LIN {X 0.009,Y -453.231,Z 340.561,A 0.000,B 0.000,C 90.000,E1 100.894} C_DIS
LIN {X 0.062,Y -474.002,Z 340.550,A 0.000,B 0.000,C 90.000,E1 99.029} C_DIS
LIN {X 0.039,Y -492.580,Z 340.542,A 0.000,B 0.000,C 90.000,E1 97.530} C_DIS
LIN {X -0.190,Y -494.914,Z 340.541,A 0.000,B 0.000,C 90.000,E1 97.352} C_DIS
LIN {X 0.008,Y -496.686,Z 340.540,A 0.000,B 0.000,C 90.000,E1 97.125} C_DIS
LIN {X -0.081,Y -498.310,Z 340.538,A 0.000,B 0.000,C 90.000,E1 96.891} C_DIS
LIN {X -0.231,Y -499.526,Z 340.537,A 0.000,B 0.000,C 90.000,E1 96.663} C_DIS
LIN {X 0.045,Y -500.998,Z 340.534,A 0.000,B 0.000,C 90.000,E1 96.144} C_DIS
LIN {X -0.171,Y -501.409,Z 340.531,A 0.000,B 0.000,C 90.000,E1 95.682} C_DIS
LIN {X 0.120,Y -500.821,Z 340.529,A 0.000,B 0.000,C 90.000,E1 95.163} C_DIS
LIN {X -0.087,Y -499.136,Z 340.526,A 0.000,B 0.000,C 90.000,E1 94.702} C_DIS
LIN {X -0.213,Y -497.782,Z 340.525,A 0.000,B 0.000,C 90.000,E1 94.473} C_DIS
LIN {X -0.069,Y -492.467,Z 340.521,A 0.000,B 0.000,C 90.000,E1 93.726} C_DIS
LIN {X -0.123,Y -484.683,Z 340.515,A 0.000,B 0.000,C 90.000,E1 92.751} C_DIS
LIN {X 0.233,Y -466.512,Z 340.503,A 0.000,B 0.000,C 90.000,E1 90.458} C_DIS
LIN {X 0.098,Y -445.860,Z 340.487,A 0.000,B 0.000,C 90.000,E1 87.650} C_DIS
LIN {X -0.176,Y -427.360,Z 340.471,A 0.000,B 0.000,C 90.000,E1 84.780} C_DIS
LIN {X 0.063,Y -409.042,Z 340.453,A 0.000,B 0.000,C 90.000,E1 81.489} C_DIS
LIN {X 0.021,Y -396.047,Z 340.439,A 0.000,B 0.000,C 90.000,E1 78.993} C_DIS
LIN {X 0.024,Y -387.321,Z 340.429,A 0.000,B 0.000,C 90.000,E1 77.297} C_DIS
LIN {X 0.089,Y -374.251,Z 340.415,A 0.000,B 0.000,C 90.000,E1 74.700} C_DIS
LIN {X -0.037,Y -364.049,Z 340.404,A 0.000,B 0.000,C 90.000,E1 72.670} C_DIS
LIN {X -0.149,Y -353.844,Z 340.392,A 0.000,B 0.000,C 90.000,E1 70.604} C_DIS
LIN {X 0.016,Y -340.830,Z 340.377,A 0.000,B 0.000,C 90.000,E1 67.847} C_DIS
LIN {X 0.116,Y -331.356,Z 340.365,A 0.000,B 0.000,C 90.000,E1 65.665} C_DIS
LIN {X -0.087,Y -318.001,Z 340.346,A 0.000,B 0.000,C 90.000,E1 62.231} C_DIS
LIN {X -0.032,Y -306.589,Z 340.328,A 0.000,B 0.000,C 90.000,E1 58.997} C_DIS
LIN {X -0.090,Y -295.955,Z 340.309,A 0.000,B 0.000,C 90.000,E1 55.722} C_DIS
LIN {X 0.040,Y -286.100,Z 340.291,A 0.000,B 0.000,C 90.000,E1 52.351} C_DIS
LIN {X 0.082,Y -278.584,Z 340.276,A 0.000,B 0.000,C 90.000,E1 49.622} C_DIS
LIN {X 0.101,Y -272.888,Z 340.264,A 0.000,B 0.000,C 90.000,E1 47.553} C_DIS
LIN {X 0.135,Y -265.279,Z 340.249,A 0.000,B 0.000,C 90.000,E1 44.757} C_DIS
LIN {X -0.099,Y -259.648,Z 340.237,A 0.000,B 0.000,C 90.000,E1 42.690} C_DIS
LIN {X -0.055,Y -253.941,Z 340.225,A 0.000,B 0.000,C 90.000,E1 40.539} C_DIS
LIN {X -0.091,Y -248.138,Z 340.213,A 0.000,B 0.000,C 90.000,E1 38.382} C_DIS
LIN {X -0.010,Y -240.251,Z 340.197,A 0.000,B 0.000,C 90.000,E1 35.438} C_DIS
LIN {X -0.017,Y -232.499,Z 340.180,A 0.000,B 0.000,C 90.000,E1 32.467} C_DIS
LIN {X -0.049,Y -223.369,Z 340.159,A 0.000,B 0.000,C 90.000,E1 28.693} C_DIS
LIN {X 0.043,Y -216.611,Z 340.142,A 0.000,B 0.000,C 90.000,E1 25.591} C_DIS
LIN {X 0.076,Y -210.503,Z 340.125,A 0.000,B 0.000,C 90.000,E1 22.461} C_DIS
LIN {X -0.008,Y -205.261,Z 340.107,A 0.000,B 0.000,C 90.000,E1 19.322} C_DIS
LIN {X 0.011,Y -199.604,Z 340.085,A 0.000,B 0.000,C 90.000,E1 15.315} C_DIS
LIN {X 0.091,Y -195.082,Z 340.063,A 0.000,B 0.000,C 90.000,E1 11.243} C_DIS
LIN {X -0.003,Y -191.668,Z 340.040,A 0.000,B 0.000,C 90.000,E1 7.182} C_DIS
LIN {X -0.072,Y -188.853,Z 340.008,A 0.000,B 0.000,C 90.000,E1 1.432} C_DIS
LIN {X 0.006,Y -189.839,Z 339.938,A 0.000,B 0.000,C 90.000,E1 348.757} C_DIS
LIN {X 0.053,Y -192.868,Z 339.910,A 0.000,B 0.000,C 90.000,E1 343.795} C_DIS
LIN {X 0.056,Y -196.554,Z 339.887,A 0.000,B 0.000,C 90.000,E1 339.699} C_DIS
LIN {X -0.036,Y -201.292,Z 339.865,A 0.000,B 0.000,C 90.000,E1 335.665} C_DIS
LIN {X -0.008,Y -207.084,Z 339.842,A 0.000,B 0.000,C 90.000,E1 331.641} C_DIS
LIN {X 0.024,Y -212.411,Z 339.825,A 0.000,B 0.000,C 90.000,E1 328.456} C_DIS
LIN {X -0.067,Y -219.844,Z 339.803,A 0.000,B 0.000,C 90.000,E1 324.562} C_DIS
LIN {X 0.043,Y -227.918,Z 339.782,A 0.000,B 0.000,C 90.000,E1 320.678} C_DIS
LIN {X -0.140,Y -236.318,Z 339.763,A 0.000,B 0.000,C 90.000,E1 317.310} C_DIS
LIN {X -0.079,Y -245.981,Z 339.744,A 0.000,B 0.000,C 90.000,E1 313.947} C_DIS
LIN {X 0.128,Y -256.915,Z 339.726,A 0.000,B 0.000,C 90.000,E1 310.620} C_DIS
LIN {X -0.016,Y -268.632,Z 339.708,A 0.000,B 0.000,C 90.000,E1 307.443} C_DIS
LIN {X -0.052,Y -280.119,Z 339.693,A 0.000,B 0.000,C 90.000,E1 304.659} C_DIS
LIN {X -0.018,Y -291.107,Z 339.679,A 0.000,B 0.000,C 90.000,E1 302.260} C_DIS
LIN {X -0.158,Y -306.784,Z 339.663,A 0.000,B 0.000,C 90.000,E1 299.283} C_DIS
LIN {X -0.051,Y -318.097,Z 339.652,A 0.000,B 0.000,C 90.000,E1 297.308} C_DIS
LIN {X -0.013,Y -339.341,Z 339.634,A 0.000,B 0.000,C 90.000,E1 294.131} C_DIS
LIN {X 0.012,Y -352.717,Z 339.624,A 0.000,B 0.000,C 90.000,E1 292.280} C_DIS
LIN {X -0.103,Y -375.772,Z 339.607,A 0.000,B 0.000,C 90.000,E1 289.322} C_DIS
LIN {X 0.153,Y -395.779,Z 339.594,A 0.000,B 0.000,C 90.000,E1 286.985} C_DIS
LIN {X 0.143,Y -408.300,Z 339.587,A 0.000,B 0.000,C 90.000,E1 285.607} C_DIS
LIN {X -0.126,Y -423.347,Z 339.578,A 0.000,B 0.000,C 90.000,E1 284.008} C_DIS
LIN {X 0.082,Y -430.579,Z 339.573,A 0.000,B 0.000,C 90.000,E1 283.175} C_DIS
LIN {X 0.206,Y -437.414,Z 339.569,A 0.000,B 0.000,C 90.000,E1 282.355} C_DIS
LIN {X 0.175,Y -445.719,Z 339.563,A 0.000,B 0.000,C 90.000,E1 281.299} C_DIS
LIN {X 0.156,Y -453.343,Z 339.557,A 0.000,B 0.000,C 90.000,E1 280.254} C_DIS
LIN {X -0.223,Y -460.409,Z 339.551,A 0.000,B 0.000,C 90.000,E1 279.265} C_DIS
LIN {X 0.159,Y -468.590,Z 339.544,A 0.000,B 0.000,C 90.000,E1 277.936} C_DIS
LIN {X -0.059,Y -474.516,Z 339.539,A 0.000,B 0.000,C 90.000,E1 276.947} C_DIS
LIN {X 0.199,Y -479.773,Z 339.533,A 0.000,B 0.000,C 90.000,E1 275.910} C_DIS
LIN {X -0.127,Y -482.067,Z 339.530,A 0.000,B 0.000,C 90.000,E1 275.448} C_DIS
LIN {X -0.003,Y -484.044,Z 339.527,A 0.000,B 0.000,C 90.000,E1 274.935} C_DIS
LIN {X 0.172,Y -485.593,Z 339.525,A 0.000,B 0.000,C 90.000,E1 274.416} C_DIS
LIN {X -0.129,Y -486.743,Z 339.522,A 0.000,B 0.000,C 90.000,E1 273.955} C_DIS
LIN {X 0.031,Y -487.515,Z 339.519,A 0.000,B 0.000,C 90.000,E1 273.440} C_DIS
LIN {X 0.229,Y -487.879,Z 339.516,A 0.000,B 0.000,C 90.000,E1 272.922} C_DIS
LIN {X -0.083,Y -487.951,Z 339.514,A 0.000,B 0.000,C 90.000,E1 272.465} C_DIS
LIN {X -0.193,Y -487.478,Z 339.508,A 0.000,B 0.000,C 90.000,E1 271.489} C_DIS
LIN {X -0.012,Y -486.912,Z 339.505,A 0.000,B 0.000,C 90.000,E1 270.974} C_DIS
LIN {X 0.167,Y -486.115,Z 339.503,A 0.000,B 0.000,C 90.000,E1 270.458} C_DIS
LIN {X -0.142,Y -484.938,Z 339.500,A 0.000,B 0.000,C 90.000,E1 270.000} C_DIS
LIN {X 0.030,Y -483.269,Z 339.497,A 0.000,B 0.000,C 90.000,E1 269.484} C_DIS
LIN {X -0.129,Y -482.227,Z 339.496,A 0.000,B 0.000,C 90.000,E1 269.255} C_DIS
LIN {X 0.026,Y -479.578,Z 339.493,A 0.000,B 0.000,C 90.000,E1 268.740} C_DIS
LIN {X 0.163,Y -476.054,Z 339.490,A 0.000,B 0.000,C 90.000,E1 268.224} C_DIS
LIN {X 0.006,Y -473.958,Z 339.489,A 0.000,B 0.000,C 90.000,E1 267.993} C_DIS
LIN {X 0.114,Y -468.786,Z 339.486,A 0.000,B 0.000,C 90.000,E1 267.478} C_DIS
LIN {X 0.067,Y -465.947,Z 339.485,A 0.000,B 0.000,C 90.000,E1 267.249} C_DIS
LIN {X -0.155,Y -459.544,Z 339.482,A 0.000,B 0.000,C 90.000,E1 266.846} C_DIS
LIN {X 0.221,Y -452.496,Z 339.480,A 0.000,B 0.000,C 90.000,E1 266.445} C_DIS
LIN {X -0.155,Y -445.052,Z 339.479,A 0.000,B 0.000,C 90.000,E1 266.216} C_DIS
LIN {X -0.036,Y -437.239,Z 339.478,A 0.000,B 0.000,C 90.000,E1 265.988} C_DIS
LIN {X 0.127,Y -428.216,Z 339.477,A 0.000,B 0.000,C 90.000,E1 265.812} C_DIS
LIN {X 0.103,Y -421.480,Z 339.477,A 0.000,B 0.000,C 90.000,E1 265.755} C_DIS
LIN {X -0.019,Y -417.651,Z 339.476,A 0.000,B 0.000,C 90.000,E1 265.755} C_DIS
LIN {X -0.034,Y -180.912,Z 339.476,A 0.000,B 0.000,C 90.000,E1 265.755} C_DIS
LIN {X 0.074,Y -180.824,Z 339.471,A 0.000,B 0.000,C 90.000,E1 264.837} C_DIS
LIN {X -0.026,Y -178.929,Z 339.443,A 0.000,B 0.000,C 90.000,E1 259.803} C_DIS
LIN {X 0.012,Y -175.976,Z 339.415,A 0.000,B 0.000,C 90.000,E1 254.700} C_DIS
LIN {X -0.043,Y -175.465,Z 339.410,A 0.000,B 0.000,C 90.000,E1 253.866} C_DIS
LIN {X 0.014,Y -172.215,Z 339.387,A 0.000,B 0.000,C 90.000,E1 249.571} C_DIS
LIN {X -0.009,Y -171.691,Z 339.382,A 0.000,B 0.000,C 90.000,E1 248.720} C_DIS
LIN {X -0.019,Y -167.917,Z 339.358,A 0.000,B 0.000,C 90.000,E1 244.409} C_DIS
LIN {X -0.001,Y -166.660,Z 339.348,A 0.000,B 0.000,C 90.000,E1 242.666} C_DIS
LIN {X -0.084,Y -162.643,Z 339.324,A 0.000,B 0.000,C 90.000,E1 238.329} C_DIS
LIN {X -0.022,Y -161.331,Z 339.314,A 0.000,B 0.000,C 90.000,E1 236.548} C_DIS
LIN {X 0.021,Y -157.327,Z 339.290,A 0.000,B 0.000,C 90.000,E1 232.110} C_DIS
LIN {X -0.045,Y -155.308,Z 339.275,A 0.000,B 0.000,C 90.000,E1 229.461} C_DIS
LIN {X -0.007,Y -151.666,Z 339.250,A 0.000,B 0.000,C 90.000,E1 224.960} C_DIS
LIN {X 0.037,Y -150.532,Z 339.240,A 0.000,B 0.000,C 90.000,E1 223.137} C_DIS
LIN {X -0.033,Y -147.257,Z 339.215,A 0.000,B 0.000,C 90.000,E1 218.624} C_DIS
LIN {X 0.024,Y -145.283,Z 339.194,A 0.000,B 0.000,C 90.000,E1 214.945} C_DIS
LIN {X 0.058,Y -142.385,Z 339.164,A 0.000,B 0.000,C 90.000,E1 209.411} C_DIS
LIN {X -0.020,Y -141.362,Z 339.148,A 0.000,B 0.000,C 90.000,E1 206.668} C_DIS
LIN {X -0.042,Y -139.343,Z 339.112,A 0.000,B 0.000,C 90.000,E1 200.174} C_DIS
LIN {X -0.036,Y -139.012,Z 339.102,A 0.000,B 0.000,C 90.000,E1 198.308} C_DIS
LIN {X -0.041,Y -138.341,Z 339.055,A 0.000,B 0.000,C 90.000,E1 189.905} C_DIS
LIN {X -0.021,Y -139.398,Z 339.008,A 0.000,B 0.000,C 90.000,E1 181.489} C_DIS
LIN {X 0.032,Y -141.300,Z 338.972,A 0.000,B 0.000,C 90.000,E1 174.951} C_DIS
LIN {X -0.010,Y -142.662,Z 338.957,A 0.000,B 0.000,C 90.000,E1 172.186} C_DIS
LIN {X -0.061,Y -145.008,Z 338.931,A 0.000,B 0.000,C 90.000,E1 167.589} C_DIS
LIN {X -0.071,Y -147.634,Z 338.911,A 0.000,B 0.000,C 90.000,E1 163.921} C_DIS
LIN {X 0.007,Y -150.265,Z 338.890,A 0.000,B 0.000,C 90.000,E1 160.242} C_DIS
LIN {X 0.020,Y -153.664,Z 338.870,A 0.000,B 0.000,C 90.000,E1 156.613} C_DIS
LIN {X 0.076,Y -157.079,Z 338.850,A 0.000,B 0.000,C 90.000,E1 152.999} C_DIS
LIN {X 0.015,Y -161.214,Z 338.830,A 0.000,B 0.000,C 90.000,E1 149.459} C_DIS
LIN {X -0.037,Y -163.303,Z 338.821,A 0.000,B 0.000,C 90.000,E1 147.709} C_DIS
LIN {X -0.028,Y -167.752,Z 338.801,A 0.000,B 0.000,C 90.000,E1 144.196} C_DIS
LIN {X -0.009,Y -171.569,Z 338.787,A 0.000,B 0.000,C 90.000,E1 141.582} C_DIS
LIN {X -0.075,Y -176.516,Z 338.767,A 0.000,B 0.000,C 90.000,E1 138.162} C_DIS
LIN {X 0.050,Y -180.814,Z 338.753,A 0.000,B 0.000,C 90.000,E1 135.567} C_DIS
LIN {X 0.035,Y -186.222,Z 338.735,A 0.000,B 0.000,C 90.000,E1 132.204} C_DIS
LIN {X -0.027,Y -190.859,Z 338.721,A 0.000,B 0.000,C 90.000,E1 129.725} C_DIS
LIN {X 0.007,Y -196.621,Z 338.702,A 0.000,B 0.000,C 90.000,E1 126.423} C_DIS
LIN {X 0.100,Y -200.747,Z 338.691,A 0.000,B 0.000,C 90.000,E1 124.326} C_DIS
LIN {X 0.115,Y -300.828,Z 338.691,A 0.000,B 0.000,C 90.000,E1 124.326} C_DIS
LIN {X -0.175,Y -306.487,Z 338.690,A 0.000,B 0.000,C 90.000,E1 124.199} C_DIS
LIN {X -0.039,Y -308.951,Z 338.689,A 0.000,B 0.000,C 90.000,E1 123.992} C_DIS
LIN {X -0.176,Y -312.801,Z 338.686,A 0.000,B 0.000,C 90.000,E1 123.579} C_DIS
LIN {X -0.045,Y -314.697,Z 338.685,A 0.000,B 0.000,C 90.000,E1 123.245} C_DIS
LIN {X -0.176,Y -316.191,Z 338.683,A 0.000,B 0.000,C 90.000,E1 122.959} C_DIS
LIN {X 0.029,Y -329.310,Z 338.663,A 0.000,B 0.000,C 90.000,E1 119.411} C_DIS
LIN {X -0.078,Y -341.472,Z 338.648,A 0.000,B 0.000,C 90.000,E1 116.616} C_DIS
LIN {X -0.012,Y -353.536,Z 338.634,A 0.000,B 0.000,C 90.000,E1 114.155} C_DIS
LIN {X -0.113,Y -366.874,Z 338.621,A 0.000,B 0.000,C 90.000,E1 111.770} C_DIS
LIN {X 0.053,Y -381.582,Z 338.608,A 0.000,B 0.000,C 90.000,E1 109.396} C_DIS
LIN {X 0.113,Y -397.769,Z 338.595,A 0.000,B 0.000,C 90.000,E1 107.094} C_DIS
LIN {X -0.164,Y -415.556,Z 338.583,A 0.000,B 0.000,C 90.000,E1 104.898} C_DIS
LIN {X 0.040,Y -435.006,Z 338.571,A 0.000,B 0.000,C 90.000,E1 102.703} C_DIS
LIN {X -0.132,Y -455.300,Z 338.559,A 0.000,B 0.000,C 90.000,E1 100.715} C_DIS
LIN {X -0.032,Y -476.123,Z 338.549,A 0.000,B 0.000,C 90.000,E1 98.859} C_DIS
LIN {X 0.140,Y -494.540,Z 338.541,A 0.000,B 0.000,C 90.000,E1 97.352} C_DIS
LIN {X -0.157,Y -496.447,Z 338.540,A 0.000,B 0.000,C 90.000,E1 97.182} C_DIS
LIN {X 0.247,Y -498.182,Z 338.538,A 0.000,B 0.000,C 90.000,E1 96.891} C_DIS
LIN {X 0.097,Y -499.483,Z 338.537,A 0.000,B 0.000,C 90.000,E1 96.663} C_DIS
LIN {X -0.125,Y -501.090,Z 338.534,A 0.000,B 0.000,C 90.000,E1 96.201} C_DIS
LIN {X 0.159,Y -501.614,Z 338.532,A 0.000,B 0.000,C 90.000,E1 95.682} C_DIS
LIN {X -0.050,Y -501.141,Z 338.529,A 0.000,B 0.000,C 90.000,E1 95.220} C_DIS
LIN {X 0.241,Y -499.590,Z 338.526,A 0.000,B 0.000,C 90.000,E1 94.702} C_DIS
LIN {X 0.116,Y -498.324,Z 338.525,A 0.000,B 0.000,C 90.000,E1 94.473} C_DIS
LIN {X -0.231,Y -493.062,Z 338.521,A 0.000,B 0.000,C 90.000,E1 93.784} C_DIS
LIN {X 0.207,Y -485.329,Z 338.515,A 0.000,B 0.000,C 90.000,E1 92.751} C_DIS
LIN {X 0.101,Y -467.113,Z 338.503,A 0.000,B 0.000,C 90.000,E1 90.516} C_DIS
LIN {X -0.010,Y -446.408,Z 338.487,A 0.000,B 0.000,C 90.000,E1 87.707} C_DIS
LIN {X 0.164,Y -427.828,Z 338.471,A 0.000,B 0.000,C 90.000,E1 84.780} C_DIS
LIN {X 0.000,Y -409.501,Z 338.453,A 0.000,B 0.000,C 90.000,E1 81.546} C_DIS
LIN {X -0.025,Y -396.518,Z 338.439,A 0.000,B 0.000,C 90.000,E1 79.050} C_DIS
LIN {X -0.011,Y -387.800,Z 338.430,A 0.000,B 0.000,C 90.000,E1 77.353} C_DIS
LIN {X 0.072,Y -374.714,Z 338.415,A 0.000,B 0.000,C 90.000,E1 74.755} C_DIS
LIN {X -0.040,Y -364.517,Z 338.404,A 0.000,B 0.000,C 90.000,E1 72.725} C_DIS
LIN {X 0.195,Y -354.305,Z 338.392,A 0.000,B 0.000,C 90.000,E1 70.604} C_DIS
LIN {X -0.083,Y -341.288,Z 338.377,A 0.000,B 0.000,C 90.000,E1 67.922} C_DIS
LIN {X 0.022,Y -331.789,Z 338.365,A 0.000,B 0.000,C 90.000,E1 65.741} C_DIS
LIN {X -0.023,Y -318.435,Z 338.346,A 0.000,B 0.000,C 90.000,E1 62.281} C_DIS
LIN {X -0.064,Y -305.897,Z 338.326,A 0.000,B 0.000,C 90.000,E1 58.742} C_DIS
LIN {X 0.031,Y -294.336,Z 338.306,A 0.000,B 0.000,C 90.000,E1 55.102} C_DIS
LIN {X 0.049,Y -284.581,Z 338.288,A 0.000,B 0.000,C 90.000,E1 51.743} C_DIS
LIN {X 0.057,Y -277.079,Z 338.272,A 0.000,B 0.000,C 90.000,E1 49.013} C_DIS
LIN {X 0.048,Y -271.336,Z 338.261,A 0.000,B 0.000,C 90.000,E1 46.944} C_DIS
LIN {X -0.146,Y -263.784,Z 338.245,A 0.000,B 0.000,C 90.000,E1 44.190} C_DIS
LIN {X 0.047,Y -256.224,Z 338.230,A 0.000,B 0.000,C 90.000,E1 41.310} C_DIS
LIN {X -0.138,Y -250.470,Z 338.218,A 0.000,B 0.000,C 90.000,E1 39.197} C_DIS
LIN {X -0.047,Y -244.568,Z 338.205,A 0.000,B 0.000,C 90.000,E1 36.996} C_DIS
LIN {X -0.007,Y -236.727,Z 338.189,A 0.000,B 0.000,C 90.000,E1 34.040} C_DIS
LIN {X 0.124,Y -227.275,Z 338.168,A 0.000,B 0.000,C 90.000,E1 30.256} C_DIS
LIN {X -0.090,Y -218.546,Z 338.147,A 0.000,B 0.000,C 90.000,E1 26.488} C_DIS
LIN {X 0.082,Y -212.229,Z 338.130,A 0.000,B 0.000,C 90.000,E1 23.334} C_DIS
LIN {X 0.045,Y -206.750,Z 338.112,A 0.000,B 0.000,C 90.000,E1 20.194} C_DIS
LIN {X 0.043,Y -200.875,Z 338.090,A 0.000,B 0.000,C 90.000,E1 16.205} C_DIS
LIN {X -0.060,Y -196.971,Z 338.072,A 0.000,B 0.000,C 90.000,E1 13.008} C_DIS
LIN {X 0.006,Y -193.094,Z 338.050,A 0.000,B 0.000,C 90.000,E1 8.916} C_DIS
LIN {X -0.079,Y -189.956,Z 338.022,A 0.000,B 0.000,C 90.000,E1 4.012} C_DIS
LIN {X -0.027,Y -190.716,Z 337.928,A 0.000,B 0.000,C 90.000,E1 347.117} C_DIS
LIN {X -0.032,Y -194.238,Z 337.901,A 0.000,B 0.000,C 90.000,E1 342.181} C_DIS
LIN {X -0.046,Y -198.343,Z 337.878,A 0.000,B 0.000,C 90.000,E1 338.103} C_DIS
LIN {X 0.077,Y -203.519,Z 337.856,A 0.000,B 0.000,C 90.000,E1 334.024} C_DIS
LIN {X 0.003,Y -209.629,Z 337.834,A 0.000,B 0.000,C 90.000,E1 330.049} C_DIS
LIN {X 0.078,Y -216.752,Z 337.812,A 0.000,B 0.000,C 90.000,E1 326.087} C_DIS
LIN {X 0.143,Y -224.531,Z 337.790,A 0.000,B 0.000,C 90.000,E1 322.190} C_DIS
LIN {X -0.029,Y -231.488,Z 337.773,A 0.000,B 0.000,C 90.000,E1 319.175} C_DIS
LIN {X 0.085,Y -239.347,Z 337.756,A 0.000,B 0.000,C 90.000,E1 316.134} C_DIS
LIN {X -0.097,Y -249.498,Z 337.738,A 0.000,B 0.000,C 90.000,E1 312.852} C_DIS
LIN {X 0.041,Y -260.745,Z 337.720,A 0.000,B 0.000,C 90.000,E1 309.564} C_DIS
LIN {X 0.054,Y -272.865,Z 337.702,A 0.000,B 0.000,C 90.000,E1 306.377} C_DIS
LIN {X -0.072,Y -286.402,Z 337.685,A 0.000,B 0.000,C 90.000,E1 303.293} C_DIS
LIN {X -0.039,Y -301.568,Z 337.668,A 0.000,B 0.000,C 90.000,E1 300.256} C_DIS
LIN {X -0.080,Y -316.345,Z 337.653,A 0.000,B 0.000,C 90.000,E1 297.641} C_DIS
LIN {X -0.093,Y -337.413,Z 337.636,A 0.000,B 0.000,C 90.000,E1 294.463} C_DIS
LIN {X 0.034,Y -350.753,Z 337.626,A 0.000,B 0.000,C 90.000,E1 292.589} C_DIS
LIN {X 0.088,Y -368.997,Z 337.612,A 0.000,B 0.000,C 90.000,E1 290.174} C_DIS
LIN {X -0.144,Y -395.974,Z 337.595,A 0.000,B 0.000,C 90.000,E1 287.040} C_DIS
LIN {X 0.066,Y -408.645,Z 337.587,A 0.000,B 0.000,C 90.000,E1 285.607} C_DIS
LIN {X -0.243,Y -423.658,Z 337.578,A 0.000,B 0.000,C 90.000,E1 284.008} C_DIS
LIN {X -0.083,Y -430.903,Z 337.573,A 0.000,B 0.000,C 90.000,E1 283.175} C_DIS
LIN {X 0.040,Y -437.677,Z 337.569,A 0.000,B 0.000,C 90.000,E1 282.355} C_DIS
LIN {X 0.010,Y -445.911,Z 337.563,A 0.000,B 0.000,C 90.000,E1 281.299} C_DIS
LIN {X -0.011,Y -453.477,Z 337.557,A 0.000,B 0.000,C 90.000,E1 280.254} C_DIS
LIN {X 0.064,Y -460.491,Z 337.551,A 0.000,B 0.000,C 90.000,E1 279.208} C_DIS
LIN {X -0.010,Y -468.644,Z 337.544,A 0.000,B 0.000,C 90.000,E1 277.936} C_DIS
LIN {X 0.241,Y -474.530,Z 337.538,A 0.000,B 0.000,C 90.000,E1 276.891} C_DIS
LIN {X 0.027,Y -479.776,Z 337.533,A 0.000,B 0.000,C 90.000,E1 275.910} C_DIS
LIN {X 0.180,Y -482.032,Z 337.530,A 0.000,B 0.000,C 90.000,E1 275.391} C_DIS
LIN {X -0.177,Y -483.995,Z 337.527,A 0.000,B 0.000,C 90.000,E1 274.935} C_DIS
LIN {X -0.003,Y -485.531,Z 337.525,A 0.000,B 0.000,C 90.000,E1 274.416} C_DIS
LIN {X 0.181,Y -486.657,Z 337.522,A 0.000,B 0.000,C 90.000,E1 273.898} C_DIS
LIN {X -0.144,Y -487.374,Z 337.519,A 0.000,B 0.000,C 90.000,E1 273.440} C_DIS
LIN {X 0.052,Y -487.715,Z 337.516,A 0.000,B 0.000,C 90.000,E1 272.922} C_DIS
LIN {X 0.227,Y -487.811,Z 337.514,A 0.000,B 0.000,C 90.000,E1 272.407} C_DIS
LIN {X 0.115,Y -487.312,Z 337.508,A 0.000,B 0.000,C 90.000,E1 271.432} C_DIS
LIN {X -0.193,Y -486.761,Z 337.505,A 0.000,B 0.000,C 90.000,E1 270.974} C_DIS
LIN {X -0.014,Y -485.983,Z 337.503,A 0.000,B 0.000,C 90.000,E1 270.458} C_DIS
LIN {X 0.162,Y -484.816,Z 337.500,A 0.000,B 0.000,C 90.000,E1 269.943} C_DIS
LIN {X -0.151,Y -483.152,Z 337.497,A 0.000,B 0.000,C 90.000,E1 269.484} C_DIS
LIN {X 0.012,Y -480.854,Z 337.494,A 0.000,B 0.000,C 90.000,E1 268.969} C_DIS
LIN {X 0.157,Y -477.831,Z 337.492,A 0.000,B 0.000,C 90.000,E1 268.453} C_DIS
LIN {X -0.174,Y -473.839,Z 337.489,A 0.000,B 0.000,C 90.000,E1 267.993} C_DIS
LIN {X -0.065,Y -468.715,Z 337.486,A 0.000,B 0.000,C 90.000,E1 267.478} C_DIS
LIN {X -0.193,Y -462.406,Z 337.483,A 0.000,B 0.000,C 90.000,E1 267.020} C_DIS
LIN {X 0.077,Y -459.185,Z 337.482,A 0.000,B 0.000,C 90.000,E1 266.788} C_DIS
LIN {X -0.003,Y -452.049,Z 337.480,A 0.000,B 0.000,C 90.000,E1 266.445} C_DIS
LIN {X 0.085,Y -444.599,Z 337.479,A 0.000,B 0.000,C 90.000,E1 266.159} C_DIS
LIN {X -0.225,Y -436.603,Z 337.478,A 0.000,B 0.000,C 90.000,E1 265.988} C_DIS
LIN {X -0.027,Y -427.272,Z 337.477,A 0.000,B 0.000,C 90.000,E1 265.812} C_DIS
LIN {X -0.087,Y -417.710,Z 337.476,A 0.000,B 0.000,C 90.000,E1 265.755} C_DIS
LIN {X -0.062,Y -180.911,Z 337.476,A 0.000,B 0.000,C 90.000,E1 265.755} C_DIS
LIN {X 0.029,Y -180.820,Z 337.471,A 0.000,B 0.000,C 90.000,E1 264.837} C_DIS
LIN {X -0.071,Y -178.924,Z 337.443,A 0.000,B 0.000,C 90.000,E1 259.803} C_DIS
LIN {X -0.033,Y -175.970,Z 337.415,A 0.000,B 0.000,C 90.000,E1 254.700} C_DIS
LIN {X -0.038,Y -175.453,Z 337.410,A 0.000,B 0.000,C 90.000,E1 253.850} C_DIS
LIN {X -0.029,Y -172.206,Z 337.386,A 0.000,B 0.000,C 90.000,E1 249.571} C_DIS
LIN {X -0.052,Y -171.680,Z 337.382,A 0.000,B 0.000,C 90.000,E1 248.720} C_DIS
LIN {X -0.061,Y -167.906,Z 337.358,A 0.000,B 0.000,C 90.000,E1 244.409} C_DIS
LIN {X -0.042,Y -166.647,Z 337.348,A 0.000,B 0.000,C 90.000,E1 242.666} C_DIS
LIN {X 0.012,Y -162.631,Z 337.324,A 0.000,B 0.000,C 90.000,E1 238.280} C_DIS
LIN {X 0.071,Y -161.319,Z 337.314,A 0.000,B 0.000,C 90.000,E1 236.501} C_DIS
LIN {X -0.019,Y -157.315,Z 337.289,A 0.000,B 0.000,C 90.000,E1 232.110} C_DIS
LIN {X -0.086,Y -155.295,Z 337.275,A 0.000,B 0.000,C 90.000,E1 229.461} C_DIS
LIN {X 0.060,Y -151.655,Z 337.250,A 0.000,B 0.000,C 90.000,E1 224.919} C_DIS
LIN {X -0.003,Y -150.522,Z 337.240,A 0.000,B 0.000,C 90.000,E1 223.137} C_DIS
LIN {X 0.020,Y -147.247,Z 337.214,A 0.000,B 0.000,C 90.000,E1 218.588} C_DIS
LIN {X -0.015,Y -145.272,Z 337.194,A 0.000,B 0.000,C 90.000,E1 214.945} C_DIS
LIN {X 0.019,Y -142.379,Z 337.163,A 0.000,B 0.000,C 90.000,E1 209.411} C_DIS
LIN {X 0.069,Y -141.354,Z 337.148,A 0.000,B 0.000,C 90.000,E1 206.616} C_DIS
LIN {X 0.051,Y -139.340,Z 337.112,A 0.000,B 0.000,C 90.000,E1 200.120} C_DIS
LIN {X -0.030,Y -139.008,Z 337.102,A 0.000,B 0.000,C 90.000,E1 198.290} C_DIS
LIN {X 0.058,Y -138.340,Z 337.055,A 0.000,B 0.000,C 90.000,E1 189.849} C_DIS
LIN {X -0.059,Y -139.403,Z 337.008,A 0.000,B 0.000,C 90.000,E1 181.489} C_DIS
LIN {X -0.005,Y -141.308,Z 336.972,A 0.000,B 0.000,C 90.000,E1 174.951} C_DIS
LIN {X -0.048,Y -142.668,Z 336.956,A 0.000,B 0.000,C 90.000,E1 172.186} C_DIS
LIN {X 0.073,Y -145.017,Z 336.931,A 0.000,B 0.000,C 90.000,E1 167.521} C_DIS
LIN {X 0.031,Y -147.644,Z 336.910,A 0.000,B 0.000,C 90.000,E1 163.866} C_DIS
LIN {X -0.033,Y -150.277,Z 336.890,A 0.000,B 0.000,C 90.000,E1 160.242} C_DIS
LIN {X -0.021,Y -153.681,Z 336.870,A 0.000,B 0.000,C 90.000,E1 156.613} C_DIS
LIN {X 0.035,Y -157.095,Z 336.850,A 0.000,B 0.000,C 90.000,E1 152.999} C_DIS
LIN {X -0.026,Y -161.233,Z 336.830,A 0.000,B 0.000,C 90.000,E1 149.459} C_DIS
LIN {X 0.059,Y -163.321,Z 336.820,A 0.000,B 0.000,C 90.000,E1 147.661} C_DIS
LIN {X -0.070,Y -167.772,Z 336.801,A 0.000,B 0.000,C 90.000,E1 144.196} C_DIS
LIN {X 0.082,Y -171.588,Z 336.786,A 0.000,B 0.000,C 90.000,E1 141.537} C_DIS
LIN {X 0.012,Y -176.538,Z 336.767,A 0.000,B 0.000,C 90.000,E1 138.119} C_DIS
LIN {X 0.005,Y -180.837,Z 336.753,A 0.000,B 0.000,C 90.000,E1 135.567} C_DIS
LIN {X -0.010,Y -186.247,Z 336.734,A 0.000,B 0.000,C 90.000,E1 132.204} C_DIS
LIN {X -0.073,Y -190.883,Z 336.721,A 0.000,B 0.000,C 90.000,E1 129.725} C_DIS
LIN {X -0.040,Y -196.647,Z 336.702,A 0.000,B 0.000,C 90.000,E1 126.423} C_DIS
LIN {X 0.069,Y -200.850,Z 336.691,A 0.000,B 0.000,C 90.000,E1 124.278} C_DIS
LIN {X 0.071,Y -300.665,Z 336.691,A 0.000,B 0.000,C 90.000,E1 124.278} C_DIS
LIN {X 0.041,Y -301.580,Z 336.690,A 0.000,B 0.000,C 90.000,E1 124.278} C_DIS
LIN {X 0.051,Y -306.312,Z 336.690,A 0.000,B 0.000,C 90.000,E1 124.119} C_DIS
LIN {X -0.113,Y -308.604,Z 336.689,A 0.000,B 0.000,C 90.000,E1 123.992} C_DIS
LIN {X -0.110,Y -312.476,Z 336.686,A 0.000,B 0.000,C 90.000,E1 123.579} C_DIS
LIN {X 0.103,Y -314.402,Z 336.685,A 0.000,B 0.000,C 90.000,E1 123.245} C_DIS
LIN {X 0.053,Y -315.926,Z 336.683,A 0.000,B 0.000,C 90.000,E1 122.959} C_DIS
LIN {X -0.087,Y -318.377,Z 336.680,A 0.000,B 0.000,C 90.000,E1 122.339} C_DIS
LIN {X -0.025,Y -329.126,Z 336.664,A 0.000,B 0.000,C 90.000,E1 119.461} C_DIS
LIN {X 0.157,Y -341.266,Z 336.648,A 0.000,B 0.000,C 90.000,E1 116.616} C_DIS
LIN {X -0.095,Y -353.311,Z 336.634,A 0.000,B 0.000,C 90.000,E1 114.207} C_DIS
LIN {X 0.129,Y -366.627,Z 336.621,A 0.000,B 0.000,C 90.000,E1 111.770} C_DIS
LIN {X -0.061,Y -381.312,Z 336.608,A 0.000,B 0.000,C 90.000,E1 109.450} C_DIS
LIN {X -0.019,Y -397.475,Z 336.595,A 0.000,B 0.000,C 90.000,E1 107.149} C_DIS
LIN {X 0.088,Y -415.235,Z 336.583,A 0.000,B 0.000,C 90.000,E1 104.898} C_DIS
LIN {X -0.227,Y -434.661,Z 336.571,A 0.000,B 0.000,C 90.000,E1 102.771} C_DIS
LIN {X 0.108,Y -454.946,Z 336.560,A 0.000,B 0.000,C 90.000,E1 100.715} C_DIS
LIN {X 0.197,Y -475.762,Z 336.549,A 0.000,B 0.000,C 90.000,E1 98.859} C_DIS
LIN {X -0.129,Y -494.264,Z 336.541,A 0.000,B 0.000,C 90.000,E1 97.409} C_DIS
LIN {X 0.063,Y -496.288,Z 336.540,A 0.000,B 0.000,C 90.000,E1 97.182} C_DIS
LIN {X -0.018,Y -498.108,Z 336.539,A 0.000,B 0.000,C 90.000,E1 96.947} C_DIS
LIN {X -0.161,Y -499.473,Z 336.537,A 0.000,B 0.000,C 90.000,E1 96.720} C_DIS
LIN {X 0.113,Y -501.190,Z 336.535,A 0.000,B 0.000,C 90.000,E1 96.201} C_DIS
LIN {X -0.102,Y -501.805,Z 336.532,A 0.000,B 0.000,C 90.000,E1 95.739} C_DIS
LIN {X 0.189,Y -501.421,Z 336.529,A 0.000,B 0.000,C 90.000,E1 95.220} C_DIS
LIN {X -0.017,Y -499.977,Z 336.526,A 0.000,B 0.000,C 90.000,E1 94.759} C_DIS
LIN {X -0.141,Y -498.779,Z 336.525,A 0.000,B 0.000,C 90.000,E1 94.531} C_DIS
LIN {X 0.138,Y -495.405,Z 336.522,A 0.000,B 0.000,C 90.000,E1 94.012} C_DIS
LIN {X 0.227,Y -489.833,Z 336.518,A 0.000,B 0.000,C 90.000,E1 93.269} C_DIS
LIN {X 0.142,Y -481.806,Z 336.513,A 0.000,B 0.000,C 90.000,E1 92.293} C_DIS
LIN {X -0.204,Y -457.951,Z 336.496,A 0.000,B 0.000,C 90.000,E1 89.312} C_DIS
LIN {X 0.189,Y -443.344,Z 336.485,A 0.000,B 0.000,C 90.000,E1 87.192} C_DIS
LIN {X -0.015,Y -423.471,Z 336.467,A 0.000,B 0.000,C 90.000,E1 84.033} C_DIS
LIN {X -0.087,Y -408.443,Z 336.452,A 0.000,B 0.000,C 90.000,E1 81.319} C_DIS
LIN {X -0.076,Y -395.470,Z 336.438,A 0.000,B 0.000,C 90.000,E1 78.814} C_DIS
LIN {X -0.078,Y -386.754,Z 336.428,A 0.000,B 0.000,C 90.000,E1 77.117} C_DIS
LIN {X -0.025,Y -375.108,Z 336.416,A 0.000,B 0.000,C 90.000,E1 74.810} C_DIS
LIN {X -0.122,Y -364.921,Z 336.404,A 0.000,B 0.000,C 90.000,E1 72.779} C_DIS
LIN {X 0.011,Y -354.701,Z 336.393,A 0.000,B 0.000,C 90.000,E1 70.678} C_DIS
LIN {X -0.132,Y -341.692,Z 336.378,A 0.000,B 0.000,C 90.000,E1 67.975} C_DIS
LIN {X -0.012,Y -332.176,Z 336.366,A 0.000,B 0.000,C 90.000,E1 65.793} C_DIS
LIN {X -0.183,Y -318.805,Z 336.346,A 0.000,B 0.000,C 90.000,E1 62.359} C_DIS
LIN {X -0.099,Y -307.403,Z 336.328,A 0.000,B 0.000,C 90.000,E1 59.125} C_DIS
LIN {X 0.120,Y -296.744,Z 336.310,A 0.000,B 0.000,C 90.000,E1 55.801} C_DIS
LIN {X 0.035,Y -286.843,Z 336.292,A 0.000,B 0.000,C 90.000,E1 52.477} C_DIS
LIN {X 0.102,Y -279.279,Z 336.276,A 0.000,B 0.000,C 90.000,E1 49.747} C_DIS
LIN {X -0.044,Y -273.588,Z 336.265,A 0.000,B 0.000,C 90.000,E1 47.715} C_DIS
LIN {X 0.010,Y -265.960,Z 336.250,A 0.000,B 0.000,C 90.000,E1 44.919} C_DIS
LIN {X -0.033,Y -260.331,Z 336.238,A 0.000,B 0.000,C 90.000,E1 42.813} C_DIS
LIN {X 0.018,Y -254.639,Z 336.226,A 0.000,B 0.000,C 90.000,E1 40.663} C_DIS
LIN {X -0.011,Y -248.859,Z 336.214,A 0.000,B 0.000,C 90.000,E1 38.508} C_DIS
LIN {X 0.090,Y -242.920,Z 336.202,A 0.000,B 0.000,C 90.000,E1 36.297} C_DIS
LIN {X -0.045,Y -235.119,Z 336.185,A 0.000,B 0.000,C 90.000,E1 33.372} C_DIS
LIN {X 0.041,Y -225.781,Z 336.164,A 0.000,B 0.000,C 90.000,E1 29.589} C_DIS
LIN {X -0.010,Y -218.811,Z 336.147,A 0.000,B 0.000,C 90.000,E1 26.539} C_DIS
LIN {X -0.034,Y -212.473,Z 336.130,A 0.000,B 0.000,C 90.000,E1 23.439} C_DIS
LIN {X -0.071,Y -206.980,Z 336.113,A 0.000,B 0.000,C 90.000,E1 20.301} C_DIS
LIN {X -0.072,Y -201.085,Z 336.091,A 0.000,B 0.000,C 90.000,E1 16.315} C_DIS
LIN {X 0.019,Y -197.161,Z 336.073,A 0.000,B 0.000,C 90.000,E1 13.063} C_DIS
LIN {X 0.087,Y -193.284,Z 336.050,A 0.000,B 0.000,C 90.000,E1 8.973} C_DIS
LIN {X -0.008,Y -190.135,Z 336.023,A 0.000,B 0.000,C 90.000,E1 4.073} C_DIS
LIN {X 0.045,Y -188.423,Z 335.970,A 0.000,B 0.000,C 90.000,E1 354.546} C_DIS
LIN {X -0.019,Y -190.776,Z 335.928,A 0.000,B 0.000,C 90.000,E1 347.117} C_DIS
LIN {X -0.021,Y -194.277,Z 335.901,A 0.000,B 0.000,C 90.000,E1 342.181} C_DIS
LIN {X -0.035,Y -198.366,Z 335.878,A 0.000,B 0.000,C 90.000,E1 338.103} C_DIS
LIN {X 0.090,Y -203.535,Z 335.856,A 0.000,B 0.000,C 90.000,E1 334.024} C_DIS
LIN {X 0.018,Y -209.618,Z 335.834,A 0.000,B 0.000,C 90.000,E1 330.049} C_DIS
LIN {X 0.091,Y -216.720,Z 335.812,A 0.000,B 0.000,C 90.000,E1 326.087} C_DIS
LIN {X -0.022,Y -224.475,Z 335.790,A 0.000,B 0.000,C 90.000,E1 322.236} C_DIS
LIN {X -0.018,Y -231.427,Z 335.773,A 0.000,B 0.000,C 90.000,E1 319.175} C_DIS
LIN {X 0.096,Y -239.298,Z 335.756,A 0.000,B 0.000,C 90.000,E1 316.134} C_DIS
LIN {X -0.086,Y -249.501,Z 335.738,A 0.000,B 0.000,C 90.000,E1 312.852} C_DIS
LIN {X 0.054,Y -260.771,Z 335.720,A 0.000,B 0.000,C 90.000,E1 309.564} C_DIS
LIN {X 0.068,Y -272.946,Z 335.702,A 0.000,B 0.000,C 90.000,E1 306.377} C_DIS
LIN {X -0.013,Y -284.958,Z 335.687,A 0.000,B 0.000,C 90.000,E1 303.627} C_DIS
LIN {X -0.016,Y -294.798,Z 335.676,A 0.000,B 0.000,C 90.000,E1 301.592} C_DIS
LIN {X -0.047,Y -310.859,Z 335.659,A 0.000,B 0.000,C 90.000,E1 298.615} C_DIS
LIN {X -0.075,Y -320.605,Z 335.650,A 0.000,B 0.000,C 90.000,E1 297.001} C_DIS
LIN {X 0.062,Y -339.905,Z 335.634,A 0.000,B 0.000,C 90.000,E1 294.131} C_DIS
LIN {X 0.100,Y -353.264,Z 335.624,A 0.000,B 0.000,C 90.000,E1 292.280} C_DIS
LIN {X -0.164,Y -374.040,Z 335.609,A 0.000,B 0.000,C 90.000,E1 289.631} C_DIS
LIN {X -0.097,Y -396.212,Z 335.595,A 0.000,B 0.000,C 90.000,E1 287.040} C_DIS
LIN {X 0.133,Y -408.808,Z 335.587,A 0.000,B 0.000,C 90.000,E1 285.607} C_DIS
LIN {X -0.177,Y -423.733,Z 335.578,A 0.000,B 0.000,C 90.000,E1 284.008} C_DIS
LIN {X -0.023,Y -430.972,Z 335.573,A 0.000,B 0.000,C 90.000,E1 283.175} C_DIS
LIN {X 0.101,Y -437.701,Z 335.569,A 0.000,B 0.000,C 90.000,E1 282.355} C_DIS
LIN {X 0.073,Y -445.896,Z 335.563,A 0.000,B 0.000,C 90.000,E1 281.299} C_DIS
LIN {X 0.054,Y -453.447,Z 335.557,A 0.000,B 0.000,C 90.000,E1 280.254} C_DIS
LIN {X 0.128,Y -460.393,Z 335.551,A 0.000,B 0.000,C 90.000,E1 279.208} C_DIS
LIN {X 0.054,Y -468.504,Z 335.544,A 0.000,B 0.000,C 90.000,E1 277.936} C_DIS
LIN {X -0.166,Y -474.394,Z 335.538,A 0.000,B 0.000,C 90.000,E1 276.947} C_DIS
LIN {X -0.243,Y -478.413,Z 335.534,A 0.000,B 0.000,C 90.000,E1 276.201} C_DIS
LIN {X 0.241,Y -481.900,Z 335.530,A 0.000,B 0.000,C 90.000,E1 275.391} C_DIS
LIN {X -0.116,Y -483.846,Z 335.527,A 0.000,B 0.000,C 90.000,E1 274.935} C_DIS
LIN {X 0.058,Y -485.389,Z 335.525,A 0.000,B 0.000,C 90.000,E1 274.416} C_DIS
LIN {X 0.241,Y -486.497,Z 335.522,A 0.000,B 0.000,C 90.000,E1 273.898} C_DIS
LIN {X -0.086,Y -487.211,Z 335.519,A 0.000,B 0.000,C 90.000,E1 273.440} C_DIS
LIN {X 0.110,Y -487.579,Z 335.516,A 0.000,B 0.000,C 90.000,E1 272.922} C_DIS
LIN {X -0.203,Y -487.641,Z 335.514,A 0.000,B 0.000,C 90.000,E1 272.465} C_DIS
LIN {X 0.170,Y -487.146,Z 335.508,A 0.000,B 0.000,C 90.000,E1 271.432} C_DIS
LIN {X -0.138,Y -486.648,Z 335.505,A 0.000,B 0.000,C 90.000,E1 270.974} C_DIS
LIN {X 0.040,Y -485.888,Z 335.503,A 0.000,B 0.000,C 90.000,E1 270.458} C_DIS
LIN {X 0.215,Y -484.746,Z 335.500,A 0.000,B 0.000,C 90.000,E1 269.943} C_DIS
LIN {X -0.099,Y -483.145,Z 335.497,A 0.000,B 0.000,C 90.000,E1 269.484} C_DIS
LIN {X 0.064,Y -480.886,Z 335.494,A 0.000,B 0.000,C 90.000,E1 268.969} C_DIS
LIN {X 0.208,Y -477.845,Z 335.492,A 0.000,B 0.000,C 90.000,E1 268.453} C_DIS
LIN {X 0.034,Y -476.026,Z 335.490,A 0.000,B 0.000,C 90.000,E1 268.224} C_DIS
LIN {X 0.167,Y -471.532,Z 335.487,A 0.000,B 0.000,C 90.000,E1 267.707} C_DIS
LIN {X -0.014,Y -468.822,Z 335.486,A 0.000,B 0.000,C 90.000,E1 267.478} C_DIS
LIN {X -0.128,Y -462.674,Z 335.483,A 0.000,B 0.000,C 90.000,E1 267.020} C_DIS
LIN {X 0.125,Y -459.419,Z 335.482,A 0.000,B 0.000,C 90.000,E1 266.788} C_DIS
LIN {X -0.106,Y -455.670,Z 335.481,A 0.000,B 0.000,C 90.000,E1 266.617} C_DIS
LIN {X 0.118,Y -448.323,Z 335.479,A 0.000,B 0.000,C 90.000,E1 266.274} C_DIS
LIN {X -0.002,Y -440.724,Z 335.478,A 0.000,B 0.000,C 90.000,E1 266.045} C_DIS
LIN {X -0.077,Y -431.684,Z 335.477,A 0.000,B 0.000,C 90.000,E1 265.869} C_DIS
LIN {X 0.120,Y -424.683,Z 335.477,A 0.000,B 0.000,C 90.000,E1 265.755} C_DIS
LIN {X -0.154,Y -418.553,Z 335.476,A 0.000,B 0.000,C 90.000,E1 265.755} C_DIS
LIN {X 0.089,Y -180.911,Z 335.476,A 0.000,B 0.000,C 90.000,E1 265.698} C_DIS
LIN {X -0.005,Y -180.816,Z 335.471,A 0.000,B 0.000,C 90.000,E1 264.837} C_DIS
LIN {X 0.073,Y -178.919,Z 335.443,A 0.000,B 0.000,C 90.000,E1 259.746} C_DIS
LIN {X -0.018,Y -175.965,Z 335.415,A 0.000,B 0.000,C 90.000,E1 254.685} C_DIS
LIN {X 0.097,Y -175.443,Z 335.410,A 0.000,B 0.000,C 90.000,E1 253.795} C_DIS
LIN {X -0.061,Y -172.199,Z 335.386,A 0.000,B 0.000,C 90.000,E1 249.571} C_DIS
LIN {X -0.084,Y -171.673,Z 335.382,A 0.000,B 0.000,C 90.000,E1 248.720} C_DIS
LIN {X -0.092,Y -167.898,Z 335.358,A 0.000,B 0.000,C 90.000,E1 244.409} C_DIS
LIN {X 0.074,Y -166.638,Z 335.348,A 0.000,B 0.000,C 90.000,E1 242.615} C_DIS
LIN {X -0.018,Y -162.623,Z 335.324,A 0.000,B 0.000,C 90.000,E1 238.280} C_DIS
LIN {X 0.041,Y -161.309,Z 335.314,A 0.000,B 0.000,C 90.000,E1 236.501} C_DIS
LIN {X -0.050,Y -157.306,Z 335.289,A 0.000,B 0.000,C 90.000,E1 232.110} C_DIS
LIN {X 0.102,Y -155.284,Z 335.275,A 0.000,B 0.000,C 90.000,E1 229.380} C_DIS
LIN {X 0.031,Y -151.648,Z 335.250,A 0.000,B 0.000,C 90.000,E1 224.919} C_DIS
LIN {X -0.032,Y -150.515,Z 335.240,A 0.000,B 0.000,C 90.000,E1 223.137} C_DIS
LIN {X -0.009,Y -147.241,Z 335.214,A 0.000,B 0.000,C 90.000,E1 218.588} C_DIS
LIN {X -0.044,Y -145.265,Z 335.194,A 0.000,B 0.000,C 90.000,E1 214.945} C_DIS
LIN {X -0.010,Y -142.374,Z 335.163,A 0.000,B 0.000,C 90.000,E1 209.411} C_DIS
LIN {X 0.040,Y -141.349,Z 335.148,A 0.000,B 0.000,C 90.000,E1 206.616} C_DIS
LIN {X 0.023,Y -139.338,Z 335.112,A 0.000,B 0.000,C 90.000,E1 200.120} C_DIS
LIN {X 0.073,Y -139.005,Z 335.101,A 0.000,B 0.000,C 90.000,E1 198.236} C_DIS
LIN {X 0.030,Y -138.339,Z 335.055,A 0.000,B 0.000,C 90.000,E1 189.849} C_DIS
LIN {X 0.052,Y -139.405,Z 335.008,A 0.000,B 0.000,C 90.000,E1 181.432} C_DIS
LIN {X -0.034,Y -141.313,Z 334.972,A 0.000,B 0.000,C 90.000,E1 174.951} C_DIS
LIN {X -0.077,Y -142.672,Z 334.956,A 0.000,B 0.000,C 90.000,E1 172.186} C_DIS
LIN {X 0.044,Y -145.025,Z 334.931,A 0.000,B 0.000,C 90.000,E1 167.521} C_DIS
LIN {X 0.002,Y -147.651,Z 334.910,A 0.000,B 0.000,C 90.000,E1 163.866} C_DIS
LIN {X -0.063,Y -150.287,Z 334.890,A 0.000,B 0.000,C 90.000,E1 160.242} C_DIS
LIN {X -0.050,Y -153.692,Z 334.870,A 0.000,B 0.000,C 90.000,E1 156.613} C_DIS
LIN {X 0.005,Y -157.106,Z 334.850,A 0.000,B 0.000,C 90.000,E1 152.999} C_DIS
LIN {X -0.057,Y -161.247,Z 334.830,A 0.000,B 0.000,C 90.000,E1 149.459} C_DIS
LIN {X 0.028,Y -163.333,Z 334.820,A 0.000,B 0.000,C 90.000,E1 147.661} C_DIS
LIN {X 0.034,Y -167.788,Z 334.801,A 0.000,B 0.000,C 90.000,E1 144.149} C_DIS
LIN {X 0.050,Y -171.601,Z 334.786,A 0.000,B 0.000,C 90.000,E1 141.537} C_DIS
LIN {X 0.098,Y -176.555,Z 334.767,A 0.000,B 0.000,C 90.000,E1 138.081} C_DIS
LIN {X -0.028,Y -180.853,Z 334.753,A 0.000,B 0.000,C 90.000,E1 135.567} C_DIS
LIN {X -0.044,Y -186.265,Z 334.734,A 0.000,B 0.000,C 90.000,E1 132.204} C_DIS
LIN {X -0.107,Y -190.901,Z 334.721,A 0.000,B 0.000,C 90.000,E1 129.725} C_DIS
LIN {X 0.084,Y -196.667,Z 334.702,A 0.000,B 0.000,C 90.000,E1 126.377} C_DIS
LIN {X -0.007,Y -200.945,Z 334.690,A 0.000,B 0.000,C 90.000,E1 124.246} C_DIS
LIN {X -0.065,Y -301.019,Z 334.690,A 0.000,B 0.000,C 90.000,E1 124.246} C_DIS
LIN {X -0.116,Y -305.998,Z 334.689,A 0.000,B 0.000,C 90.000,E1 124.119} C_DIS
LIN {X -0.166,Y -308.170,Z 334.689,A 0.000,B 0.000,C 90.000,E1 123.992} C_DIS
LIN {X 0.009,Y -312.043,Z 334.687,A 0.000,B 0.000,C 90.000,E1 123.579} C_DIS
LIN {X -0.071,Y -315.552,Z 334.683,A 0.000,B 0.000,C 90.000,E1 123.038} C_DIS
LIN {X -0.015,Y -317.000,Z 334.682,A 0.000,B 0.000,C 90.000,E1 122.704} C_DIS
LIN {X -0.170,Y -328.892,Z 334.664,A 0.000,B 0.000,C 90.000,E1 119.539} C_DIS
LIN {X 0.008,Y -341.004,Z 334.648,A 0.000,B 0.000,C 90.000,E1 116.693} C_DIS
LIN {X -0.105,Y -353.023,Z 334.635,A 0.000,B 0.000,C 90.000,E1 114.259} C_DIS
LIN {X -0.031,Y -366.312,Z 334.621,A 0.000,B 0.000,C 90.000,E1 111.844} C_DIS
LIN {X -0.099,Y -380.968,Z 334.608,A 0.000,B 0.000,C 90.000,E1 109.504} C_DIS
LIN {X -0.188,Y -397.098,Z 334.596,A 0.000,B 0.000,C 90.000,E1 107.221} C_DIS
LIN {X 0.018,Y -414.823,Z 334.583,A 0.000,B 0.000,C 90.000,E1 104.954} C_DIS
LIN {X 0.104,Y -434.217,Z 334.571,A 0.000,B 0.000,C 90.000,E1 102.771} C_DIS
LIN {X -0.106,Y -454.490,Z 334.560,A 0.000,B 0.000,C 90.000,E1 100.782} C_DIS
LIN {X 0.031,Y -475.296,Z 334.550,A 0.000,B 0.000,C 90.000,E1 98.916} C_DIS
LIN {X 0.162,Y -493.855,Z 334.541,A 0.000,B 0.000,C 90.000,E1 97.409} C_DIS
LIN {X -0.140,Y -496.032,Z 334.540,A 0.000,B 0.000,C 90.000,E1 97.239} C_DIS
LIN {X -0.138,Y -497.900,Z 334.539,A 0.000,B 0.000,C 90.000,E1 97.004} C_DIS
LIN {X -0.195,Y -499.319,Z 334.538,A 0.000,B 0.000,C 90.000,E1 96.777} C_DIS
LIN {X 0.078,Y -501.216,Z 334.535,A 0.000,B 0.000,C 90.000,E1 96.258} C_DIS
LIN {X -0.139,Y -501.980,Z 334.532,A 0.000,B 0.000,C 90.000,E1 95.796} C_DIS
LIN {X 0.153,Y -501.741,Z 334.529,A 0.000,B 0.000,C 90.000,E1 95.277} C_DIS
LIN {X -0.095,Y -500.459,Z 334.527,A 0.000,B 0.000,C 90.000,E1 94.821} C_DIS
LIN {X -0.177,Y -499.363,Z 334.525,A 0.000,B 0.000,C 90.000,E1 94.588} C_DIS
LIN {X 0.197,Y -497.884,Z 334.524,A 0.000,B 0.000,C 90.000,E1 94.302} C_DIS
LIN {X 0.200,Y -490.594,Z 334.519,A 0.000,B 0.000,C 90.000,E1 93.326} C_DIS
LIN {X 0.123,Y -482.593,Z 334.513,A 0.000,B 0.000,C 90.000,E1 92.350} C_DIS
LIN {X -0.198,Y -458.654,Z 334.496,A 0.000,B 0.000,C 90.000,E1 89.370} C_DIS
LIN {X -0.044,Y -442.248,Z 334.483,A 0.000,B 0.000,C 90.000,E1 87.020} C_DIS
LIN {X 0.030,Y -424.048,Z 334.467,A 0.000,B 0.000,C 90.000,E1 84.090} C_DIS
LIN {X 0.088,Y -407.519,Z 334.451,A 0.000,B 0.000,C 90.000,E1 81.084} C_DIS
LIN {X 0.001,Y -396.013,Z 334.438,A 0.000,B 0.000,C 90.000,E1 78.870} C_DIS
LIN {X 0.009,Y -387.320,Z 334.429,A 0.000,B 0.000,C 90.000,E1 77.173} C_DIS
LIN {X 0.076,Y -375.653,Z 334.416,A 0.000,B 0.000,C 90.000,E1 74.866} C_DIS
LIN {X -0.009,Y -365.484,Z 334.405,A 0.000,B 0.000,C 90.000,E1 72.834} C_DIS
LIN {X 0.136,Y -355.275,Z 334.393,A 0.000,B 0.000,C 90.000,E1 70.732} C_DIS
LIN {X 0.010,Y -342.243,Z 334.378,A 0.000,B 0.000,C 90.000,E1 68.028} C_DIS
LIN {X 0.007,Y -332.698,Z 334.366,A 0.000,B 0.000,C 90.000,E1 65.869} C_DIS
LIN {X -0.009,Y -319.309,Z 334.347,A 0.000,B 0.000,C 90.000,E1 62.410} C_DIS
LIN {X -0.065,Y -307.909,Z 334.329,A 0.000,B 0.000,C 90.000,E1 59.203} C_DIS
LIN {X -0.083,Y -297.232,Z 334.311,A 0.000,B 0.000,C 90.000,E1 55.928} C_DIS
LIN {X 0.089,Y -287.301,Z 334.292,A 0.000,B 0.000,C 90.000,E1 52.557} C_DIS
LIN {X 0.163,Y -279.728,Z 334.277,A 0.000,B 0.000,C 90.000,E1 49.828} C_DIS
LIN {X 0.023,Y -274.014,Z 334.266,A 0.000,B 0.000,C 90.000,E1 47.796} C_DIS
LIN {X 0.084,Y -266.378,Z 334.250,A 0.000,B 0.000,C 90.000,E1 45.000} C_DIS
LIN {X -0.129,Y -260.752,Z 334.238,A 0.000,B 0.000,C 90.000,E1 42.933} C_DIS
LIN {X -0.060,Y -255.065,Z 334.227,A 0.000,B 0.000,C 90.000,E1 40.782} C_DIS
LIN {X -0.071,Y -249.311,Z 334.214,A 0.000,B 0.000,C 90.000,E1 38.624} C_DIS
LIN {X -0.004,Y -243.370,Z 334.202,A 0.000,B 0.000,C 90.000,E1 36.423} C_DIS
LIN {X 0.068,Y -235.556,Z 334.186,A 0.000,B 0.000,C 90.000,E1 33.452} C_DIS
LIN {X -0.029,Y -226.189,Z 334.165,A 0.000,B 0.000,C 90.000,E1 29.716} C_DIS
LIN {X -0.069,Y -219.166,Z 334.148,A 0.000,B 0.000,C 90.000,E1 26.668} C_DIS
LIN {X 0.114,Y -212.798,Z 334.131,A 0.000,B 0.000,C 90.000,E1 23.515} C_DIS
LIN {X -0.107,Y -207.282,Z 334.113,A 0.000,B 0.000,C 90.000,E1 20.429} C_DIS
LIN {X -0.094,Y -201.353,Z 334.091,A 0.000,B 0.000,C 90.000,E1 16.441} C_DIS
LIN {X 0.053,Y -197.411,Z 334.073,A 0.000,B 0.000,C 90.000,E1 13.175} C_DIS
LIN {X -0.098,Y -193.518,Z 334.051,A 0.000,B 0.000,C 90.000,E1 9.151} C_DIS
LIN {X 0.033,Y -190.342,Z 334.023,A 0.000,B 0.000,C 90.000,E1 4.188} C_DIS
LIN {X 0.007,Y -188.407,Z 333.979,A 0.000,B 0.000,C 90.000,E1 356.216} C_DIS
LIN {X 0.009,Y -190.424,Z 333.933,A 0.000,B 0.000,C 90.000,E1 347.937} C_DIS
LIN {X -0.057,Y -193.654,Z 333.906,A 0.000,B 0.000,C 90.000,E1 343.015} C_DIS
LIN {X 0.034,Y -197.521,Z 333.883,A 0.000,B 0.000,C 90.000,E1 338.901} C_DIS
LIN {X 0.051,Y -202.433,Z 333.860,A 0.000,B 0.000,C 90.000,E1 334.845} C_DIS
LIN {X 0.029,Y -208.313,Z 333.838,A 0.000,B 0.000,C 90.000,E1 330.845} C_DIS
LIN {X -0.053,Y -215.232,Z 333.816,A 0.000,B 0.000,C 90.000,E1 326.914} C_DIS
LIN {X 0.005,Y -222.836,Z 333.794,A 0.000,B 0.000,C 90.000,E1 323.004} C_DIS
LIN {X 0.109,Y -229.553,Z 333.777,A 0.000,B 0.000,C 90.000,E1 319.908} C_DIS
LIN {X -0.019,Y -238.219,Z 333.759,A 0.000,B 0.000,C 90.000,E1 316.539} C_DIS
LIN {X -0.071,Y -248.334,Z 333.740,A 0.000,B 0.000,C 90.000,E1 313.218} C_DIS
LIN {X 0.033,Y -259.524,Z 333.722,A 0.000,B 0.000,C 90.000,E1 309.930} C_DIS
LIN {X 0.006,Y -271.628,Z 333.704,A 0.000,B 0.000,C 90.000,E1 306.744} C_DIS
LIN {X -0.055,Y -281.966,Z 333.691,A 0.000,B 0.000,C 90.000,E1 304.326} C_DIS
LIN {X 0.020,Y -293.260,Z 333.677,A 0.000,B 0.000,C 90.000,E1 301.926} C_DIS
LIN {X -0.048,Y -309.188,Z 333.661,A 0.000,B 0.000,C 90.000,E1 298.949} C_DIS
LIN {X -0.107,Y -318.820,Z 333.652,A 0.000,B 0.000,C 90.000,E1 297.334} C_DIS
LIN {X -0.009,Y -337.982,Z 333.636,A 0.000,B 0.000,C 90.000,E1 294.463} C_DIS
LIN {X -0.172,Y -353.537,Z 333.624,A 0.000,B 0.000,C 90.000,E1 292.333} C_DIS
LIN {X -0.099,Y -374.326,Z 333.609,A 0.000,B 0.000,C 90.000,E1 289.631} C_DIS
LIN {X -0.173,Y -396.614,Z 333.595,A 0.000,B 0.000,C 90.000,E1 287.040} C_DIS
LIN {X 0.087,Y -409.100,Z 333.587,A 0.000,B 0.000,C 90.000,E1 285.607} C_DIS
LIN {X -0.226,Y -423.942,Z 333.578,A 0.000,B 0.000,C 90.000,E1 284.008} C_DIS
LIN {X 0.101,Y -433.452,Z 333.572,A 0.000,B 0.000,C 90.000,E1 282.883} C_DIS
LIN {X 0.023,Y -441.996,Z 333.566,A 0.000,B 0.000,C 90.000,E1 281.827} C_DIS
LIN {X -0.043,Y -449.813,Z 333.560,A 0.000,B 0.000,C 90.000,E1 280.782} C_DIS
LIN {X 0.067,Y -457.043,Z 333.554,A 0.000,B 0.000,C 90.000,E1 279.726} C_DIS
LIN {X -0.062,Y -465.269,Z 333.547,A 0.000,B 0.000,C 90.000,E1 278.454} C_DIS
LIN {X 0.149,Y -471.451,Z 333.541,A 0.000,B 0.000,C 90.000,E1 277.409} C_DIS
LIN {X -0.102,Y -477.096,Z 333.536,A 0.000,B 0.000,C 90.000,E1 276.429} C_DIS
LIN {X -0.153,Y -480.763,Z 333.531,A 0.000,B 0.000,C 90.000,E1 275.682} C_DIS
LIN {X -0.172,Y -483.784,Z 333.527,A 0.000,B 0.000,C 90.000,E1 274.935} C_DIS
LIN {X 0.002,Y -485.287,Z 333.525,A 0.000,B 0.000,C 90.000,E1 274.416} C_DIS
LIN {X 0.184,Y -486.400,Z 333.522,A 0.000,B 0.000,C 90.000,E1 273.898} C_DIS
LIN {X -0.143,Y -487.092,Z 333.519,A 0.000,B 0.000,C 90.000,E1 273.440} C_DIS
LIN {X 0.051,Y -487.434,Z 333.516,A 0.000,B 0.000,C 90.000,E1 272.922} C_DIS
LIN {X 0.225,Y -487.477,Z 333.514,A 0.000,B 0.000,C 90.000,E1 272.407} C_DIS
LIN {X 0.110,Y -486.966,Z 333.508,A 0.000,B 0.000,C 90.000,E1 271.432} C_DIS
LIN {X -0.199,Y -486.474,Z 333.505,A 0.000,B 0.000,C 90.000,E1 270.974} C_DIS
LIN {X -0.023,Y -485.730,Z 333.503,A 0.000,B 0.000,C 90.000,E1 270.458} C_DIS
LIN {X 0.152,Y -484.649,Z 333.500,A 0.000,B 0.000,C 90.000,E1 269.943} C_DIS
LIN {X -0.162,Y -482.985,Z 333.497,A 0.000,B 0.000,C 90.000,E1 269.484} C_DIS
LIN {X 0.000,Y -480.800,Z 333.494,A 0.000,B 0.000,C 90.000,E1 268.969} C_DIS
LIN {X 0.144,Y -477.807,Z 333.492,A 0.000,B 0.000,C 90.000,E1 268.453} C_DIS
LIN {X -0.031,Y -475.971,Z 333.490,A 0.000,B 0.000,C 90.000,E1 268.224} C_DIS
LIN {X 0.104,Y -471.475,Z 333.487,A 0.000,B 0.000,C 90.000,E1 267.707} C_DIS
LIN {X -0.078,Y -468.777,Z 333.486,A 0.000,B 0.000,C 90.000,E1 267.478} C_DIS
LIN {X -0.140,Y -465.921,Z 333.485,A 0.000,B 0.000,C 90.000,E1 267.249} C_DIS
LIN {X -0.203,Y -462.671,Z 333.483,A 0.000,B 0.000,C 90.000,E1 267.020} C_DIS
LIN {X 0.050,Y -459.406,Z 333.482,A 0.000,B 0.000,C 90.000,E1 266.788} C_DIS
LIN {X -0.065,Y -452.273,Z 333.480,A 0.000,B 0.000,C 90.000,E1 266.445} C_DIS
LIN {X -0.008,Y -444.869,Z 333.479,A 0.000,B 0.000,C 90.000,E1 266.159} C_DIS
LIN {X 0.139,Y -436.964,Z 333.477,A 0.000,B 0.000,C 90.000,E1 265.927} C_DIS
LIN {X -0.146,Y -427.671,Z 333.477,A 0.000,B 0.000,C 90.000,E1 265.812} C_DIS
LIN {X -0.167,Y -420.750,Z 333.476,A 0.000,B 0.000,C 90.000,E1 265.755} C_DIS
LIN {X 0.131,Y -416.259,Z 333.476,A 0.000,B 0.000,C 90.000,E1 265.698} C_DIS
LIN {X 0.031,Y -180.910,Z 333.476,A 0.000,B 0.000,C 90.000,E1 265.698} C_DIS
LIN {X -0.041,Y -180.812,Z 333.471,A 0.000,B 0.000,C 90.000,E1 264.837} C_DIS
LIN {X 0.035,Y -178.915,Z 333.443,A 0.000,B 0.000,C 90.000,E1 259.746} C_DIS
LIN {X -0.054,Y -175.959,Z 333.415,A 0.000,B 0.000,C 90.000,E1 254.685} C_DIS
LIN {X 0.062,Y -175.434,Z 333.410,A 0.000,B 0.000,C 90.000,E1 253.795} C_DIS
LIN {X 0.064,Y -172.192,Z 333.386,A 0.000,B 0.000,C 90.000,E1 249.518} C_DIS
LIN {X 0.041,Y -171.665,Z 333.382,A 0.000,B 0.000,C 90.000,E1 248.666} C_DIS
LIN {X 0.024,Y -167.890,Z 333.358,A 0.000,B 0.000,C 90.000,E1 244.357} C_DIS
LIN {X 0.039,Y -166.627,Z 333.348,A 0.000,B 0.000,C 90.000,E1 242.615} C_DIS
LIN {X 0.032,Y -162.613,Z 333.324,A 0.000,B 0.000,C 90.000,E1 238.250} C_DIS
LIN {X 0.007,Y -161.299,Z 333.314,A 0.000,B 0.000,C 90.000,E1 236.501} C_DIS
LIN {X 0.040,Y -157.297,Z 333.289,A 0.000,B 0.000,C 90.000,E1 232.065} C_DIS
LIN {X 0.069,Y -155.272,Z 333.274,A 0.000,B 0.000,C 90.000,E1 229.380} C_DIS
LIN {X -0.003,Y -151.638,Z 333.250,A 0.000,B 0.000,C 90.000,E1 224.919} C_DIS
LIN {X 0.045,Y -150.508,Z 333.240,A 0.000,B 0.000,C 90.000,E1 223.095} C_DIS
LIN {X 0.074,Y -147.233,Z 333.214,A 0.000,B 0.000,C 90.000,E1 218.543} C_DIS
LIN {X 0.043,Y -145.256,Z 333.194,A 0.000,B 0.000,C 90.000,E1 214.898} C_DIS
LIN {X -0.041,Y -142.369,Z 333.163,A 0.000,B 0.000,C 90.000,E1 209.411} C_DIS
LIN {X 0.079,Y -141.754,Z 333.153,A 0.000,B 0.000,C 90.000,E1 207.513} C_DIS
LIN {X 0.005,Y -139.496,Z 333.117,A 0.000,B 0.000,C 90.000,E1 201.046} C_DIS
LIN {X 0.042,Y -139.001,Z 333.101,A 0.000,B 0.000,C 90.000,E1 198.236} C_DIS
LIN {X -0.001,Y -138.338,Z 333.055,A 0.000,B 0.000,C 90.000,E1 189.849} C_DIS
LIN {X 0.021,Y -139.409,Z 333.008,A 0.000,B 0.000,C 90.000,E1 181.432} C_DIS
LIN {X -0.066,Y -141.319,Z 332.972,A 0.000,B 0.000,C 90.000,E1 174.951} C_DIS
LIN {X 0.033,Y -142.678,Z 332.956,A 0.000,B 0.000,C 90.000,E1 172.129} C_DIS
LIN {X 0.012,Y -145.033,Z 332.931,A 0.000,B 0.000,C 90.000,E1 167.521} C_DIS
LIN {X -0.031,Y -147.658,Z 332.910,A 0.000,B 0.000,C 90.000,E1 163.866} C_DIS
LIN {X 0.045,Y -150.297,Z 332.890,A 0.000,B 0.000,C 90.000,E1 160.188} C_DIS
LIN {X -0.084,Y -153.706,Z 332.870,A 0.000,B 0.000,C 90.000,E1 156.613} C_DIS
LIN {X -0.029,Y -157.119,Z 332.850,A 0.000,B 0.000,C 90.000,E1 152.999} C_DIS
LIN {X 0.047,Y -161.263,Z 332.830,A 0.000,B 0.000,C 90.000,E1 149.410} C_DIS
LIN {X -0.026,Y -164.381,Z 332.815,A 0.000,B 0.000,C 90.000,E1 146.786} C_DIS
LIN {X -0.039,Y -169.056,Z 332.796,A 0.000,B 0.000,C 90.000,E1 143.290} C_DIS
LIN {X 0.014,Y -171.617,Z 332.786,A 0.000,B 0.000,C 90.000,E1 141.537} C_DIS
LIN {X 0.061,Y -176.574,Z 332.767,A 0.000,B 0.000,C 90.000,E1 138.081} C_DIS
LIN {X -0.065,Y -180.872,Z 332.753,A 0.000,B 0.000,C 90.000,E1 135.567} C_DIS
LIN {X 0.056,Y -186.286,Z 332.734,A 0.000,B 0.000,C 90.000,E1 132.162} C_DIS
LIN {X -0.023,Y -190.921,Z 332.720,A 0.000,B 0.000,C 90.000,E1 129.688} C_DIS
LIN {X 0.045,Y -196.688,Z 332.702,A 0.000,B 0.000,C 90.000,E1 126.377} C_DIS
LIN {X -0.074,Y -201.058,Z 332.690,A 0.000,B 0.000,C 90.000,E1 124.199} C_DIS
LIN {X -0.152,Y -302.004,Z 332.690,A 0.000,B 0.000,C 90.000,E1 124.199} C_DIS
LIN {X 0.186,Y -302.969,Z 332.690,A 0.000,B 0.000,C 90.000,E1 124.119} C_DIS
LIN {X 0.201,Y -307.681,Z 332.689,A 0.000,B 0.000,C 90.000,E1 123.913} C_DIS
LIN {X -0.144,Y -310.848,Z 332.687,A 0.000,B 0.000,C 90.000,E1 123.706} C_DIS
LIN {X 0.096,Y -314.549,Z 332.684,A 0.000,B 0.000,C 90.000,E1 123.166} C_DIS
LIN {X -0.117,Y -316.254,Z 332.683,A 0.000,B 0.000,C 90.000,E1 122.880} C_DIS
LIN {X 0.004,Y -318.724,Z 332.679,A 0.000,B 0.000,C 90.000,E1 122.212} C_DIS
LIN {X 0.078,Y -329.526,Z 332.663,A 0.000,B 0.000,C 90.000,E1 119.333} C_DIS
LIN {X -0.024,Y -341.718,Z 332.647,A 0.000,B 0.000,C 90.000,E1 116.539} C_DIS
LIN {X 0.045,Y -353.815,Z 332.634,A 0.000,B 0.000,C 90.000,E1 114.079} C_DIS
LIN {X -0.192,Y -367.188,Z 332.620,A 0.000,B 0.000,C 90.000,E1 111.716} C_DIS
LIN {X 0.112,Y -381.934,Z 332.607,A 0.000,B 0.000,C 90.000,E1 109.322} C_DIS
LIN {X 0.057,Y -398.163,Z 332.595,A 0.000,B 0.000,C 90.000,E1 107.040} C_DIS
LIN {X -0.102,Y -415.994,Z 332.582,A 0.000,B 0.000,C 90.000,E1 104.828} C_DIS
LIN {X 0.030,Y -435.467,Z 332.570,A 0.000,B 0.000,C 90.000,E1 102.647} C_DIS
LIN {X -0.105,Y -455.776,Z 332.559,A 0.000,B 0.000,C 90.000,E1 100.658} C_DIS
LIN {X 0.032,Y -476.612,Z 332.549,A 0.000,B 0.000,C 90.000,E1 98.803} C_DIS
LIN {X 0.219,Y -495.080,Z 332.541,A 0.000,B 0.000,C 90.000,E1 97.296} C_DIS
LIN {X 0.031,Y -498.608,Z 332.538,A 0.000,B 0.000,C 90.000,E1 96.891} C_DIS
LIN {X -0.118,Y -499.954,Z 332.537,A 0.000,B 0.000,C 90.000,E1 96.663} C_DIS
LIN {X -0.210,Y -500.945,Z 332.536,A 0.000,B 0.000,C 90.000,E1 96.429} C_DIS
LIN {X 0.074,Y -502.046,Z 332.533,A 0.000,B 0.000,C 90.000,E1 95.910} C_DIS
LIN {X -0.137,Y -502.124,Z 332.530,A 0.000,B 0.000,C 90.000,E1 95.448} C_DIS
LIN {X 0.114,Y -501.190,Z 332.527,A 0.000,B 0.000,C 90.000,E1 94.935} C_DIS
LIN {X -0.089,Y -499.075,Z 332.525,A 0.000,B 0.000,C 90.000,E1 94.473} C_DIS
LIN {X 0.064,Y -493.879,Z 332.521,A 0.000,B 0.000,C 90.000,E1 93.726} C_DIS
LIN {X 0.022,Y -486.133,Z 332.515,A 0.000,B 0.000,C 90.000,E1 92.751} C_DIS
LIN {X 0.133,Y -469.819,Z 332.504,A 0.000,B 0.000,C 90.000,E1 90.745} C_DIS
LIN {X -0.130,Y -450.669,Z 332.490,A 0.000,B 0.000,C 90.000,E1 88.224} C_DIS
LIN {X -0.130,Y -434.990,Z 332.477,A 0.000,B 0.000,C 90.000,E1 85.869} C_DIS
LIN {X 0.046,Y -418.974,Z 332.462,A 0.000,B 0.000,C 90.000,E1 83.166} C_DIS
LIN {X -0.199,Y -405.669,Z 332.448,A 0.000,B 0.000,C 90.000,E1 80.735} C_DIS
LIN {X -0.008,Y -395.635,Z 332.438,A 0.000,B 0.000,C 90.000,E1 78.757} C_DIS
LIN {X -0.012,Y -386.934,Z 332.428,A 0.000,B 0.000,C 90.000,E1 77.061} C_DIS
LIN {X 0.040,Y -375.282,Z 332.415,A 0.000,B 0.000,C 90.000,E1 74.755} C_DIS
LIN {X -0.063,Y -365.106,Z 332.404,A 0.000,B 0.000,C 90.000,E1 72.725} C_DIS
LIN {X 0.190,Y -354.897,Z 332.392,A 0.000,B 0.000,C 90.000,E1 70.604} C_DIS
LIN {X -0.077,Y -341.879,Z 332.377,A 0.000,B 0.000,C 90.000,E1 67.922} C_DIS
LIN {X 0.022,Y -331.127,Z 332.364,A 0.000,B 0.000,C 90.000,E1 65.433} C_DIS
LIN {X -0.049,Y -317.907,Z 332.344,A 0.000,B 0.000,C 90.000,E1 61.975} C_DIS
LIN {X -0.002,Y -306.578,Z 332.326,A 0.000,B 0.000,C 90.000,E1 58.742} C_DIS
LIN {X -0.061,Y -296.029,Z 332.308,A 0.000,B 0.000,C 90.000,E1 55.468} C_DIS
LIN {X 0.007,Y -286.190,Z 332.290,A 0.000,B 0.000,C 90.000,E1 52.110} C_DIS
LIN {X 0.058,Y -278.627,Z 332.274,A 0.000,B 0.000,C 90.000,E1 49.380} C_DIS
LIN {X 0.081,Y -272.863,Z 332.263,A 0.000,B 0.000,C 90.000,E1 47.310} C_DIS
LIN {X 0.115,Y -265.254,Z 332.247,A 0.000,B 0.000,C 90.000,E1 44.514} C_DIS
LIN {X -0.121,Y -259.617,Z 332.236,A 0.000,B 0.000,C 90.000,E1 42.447} C_DIS
LIN {X -0.078,Y -253.911,Z 332.224,A 0.000,B 0.000,C 90.000,E1 40.297} C_DIS
LIN {X 0.078,Y -248.149,Z 332.212,A 0.000,B 0.000,C 90.000,E1 38.096} C_DIS
LIN {X -0.029,Y -242.218,Z 332.200,A 0.000,B 0.000,C 90.000,E1 35.931} C_DIS
LIN {X 0.015,Y -234.423,Z 332.183,A 0.000,B 0.000,C 90.000,E1 32.959} C_DIS
LIN {X -0.039,Y -225.095,Z 332.162,A 0.000,B 0.000,C 90.000,E1 29.205} C_DIS
LIN {X 0.094,Y -218.154,Z 332.145,A 0.000,B 0.000,C 90.000,E1 26.104} C_DIS
LIN {X -0.030,Y -211.899,Z 332.128,A 0.000,B 0.000,C 90.000,E1 23.025} C_DIS
LIN {X -0.072,Y -206.548,Z 332.110,A 0.000,B 0.000,C 90.000,E1 19.885} C_DIS
LIN {X -0.001,Y -201.831,Z 332.093,A 0.000,B 0.000,C 90.000,E1 16.677} C_DIS
LIN {X -0.035,Y -197.824,Z 332.075,A 0.000,B 0.000,C 90.000,E1 13.467} C_DIS
LIN {X 0.049,Y -193.881,Z 332.052,A 0.000,B 0.000,C 90.000,E1 9.378} C_DIS
LIN {X -0.008,Y -190.623,Z 332.025,A 0.000,B 0.000,C 90.000,E1 4.473} C_DIS
LIN {X 0.090,Y -188.552,Z 331.984,A 0.000,B 0.000,C 90.000,E1 357.020} C_DIS
LIN {X 0.017,Y -190.504,Z 331.933,A 0.000,B 0.000,C 90.000,E1 347.937} C_DIS
LIN {X -0.045,Y -193.718,Z 331.906,A 0.000,B 0.000,C 90.000,E1 343.015} C_DIS
LIN {X 0.048,Y -197.575,Z 331.883,A 0.000,B 0.000,C 90.000,E1 338.901} C_DIS
LIN {X 0.067,Y -202.470,Z 331.860,A 0.000,B 0.000,C 90.000,E1 334.845} C_DIS
LIN {X 0.046,Y -208.330,Z 331.838,A 0.000,B 0.000,C 90.000,E1 330.845} C_DIS
LIN {X -0.034,Y -215.228,Z 331.816,A 0.000,B 0.000,C 90.000,E1 326.914} C_DIS
LIN {X 0.025,Y -222.800,Z 331.794,A 0.000,B 0.000,C 90.000,E1 323.004} C_DIS
LIN {X 0.128,Y -229.523,Z 331.777,A 0.000,B 0.000,C 90.000,E1 319.908} C_DIS
LIN {X 0.000,Y -238.211,Z 331.759,A 0.000,B 0.000,C 90.000,E1 316.539} C_DIS
LIN {X -0.051,Y -248.347,Z 331.740,A 0.000,B 0.000,C 90.000,E1 313.218} C_DIS
LIN {X 0.055,Y -259.570,Z 331.722,A 0.000,B 0.000,C 90.000,E1 309.930} C_DIS
LIN {X 0.030,Y -271.712,Z 331.704,A 0.000,B 0.000,C 90.000,E1 306.744} C_DIS
LIN {X 0.023,Y -280.525,Z 331.693,A 0.000,B 0.000,C 90.000,E1 304.659} C_DIS
LIN {X 0.051,Y -293.421,Z 331.677,A 0.000,B 0.000,C 90.000,E1 301.926} C_DIS
LIN {X -0.010,Y -309.419,Z 331.661,A 0.000,B 0.000,C 90.000,E1 298.949} C_DIS
LIN {X -0.064,Y -319.075,Z 331.652,A 0.000,B 0.000,C 90.000,E1 297.334} C_DIS
LIN {X 0.043,Y -338.256,Z 331.636,A 0.000,B 0.000,C 90.000,E1 294.463} C_DIS
LIN {X -0.112,Y -353.808,Z 331.624,A 0.000,B 0.000,C 90.000,E1 292.333} C_DIS
LIN {X -0.199,Y -369.852,Z 331.612,A 0.000,B 0.000,C 90.000,E1 290.248} C_DIS
LIN {X -0.127,Y -394.293,Z 331.596,A 0.000,B 0.000,C 90.000,E1 287.330} C_DIS
LIN {X 0.099,Y -406.743,Z 331.588,A 0.000,B 0.000,C 90.000,E1 285.898} C_DIS
LIN {X -0.158,Y -421.394,Z 331.579,A 0.000,B 0.000,C 90.000,E1 284.300} C_DIS
LIN {X 0.221,Y -430.950,Z 331.573,A 0.000,B 0.000,C 90.000,E1 283.175} C_DIS
LIN {X -0.079,Y -437.627,Z 331.569,A 0.000,B 0.000,C 90.000,E1 282.411} C_DIS
LIN {X -0.201,Y -445.737,Z 331.563,A 0.000,B 0.000,C 90.000,E1 281.366} C_DIS
LIN {X -0.139,Y -453.233,Z 331.557,A 0.000,B 0.000,C 90.000,E1 280.310} C_DIS
LIN {X -0.072,Y -460.113,Z 331.551,A 0.000,B 0.000,C 90.000,E1 279.265} C_DIS
LIN {X -0.155,Y -468.113,Z 331.544,A 0.000,B 0.000,C 90.000,E1 277.992} C_DIS
LIN {X 0.087,Y -474.008,Z 331.539,A 0.000,B 0.000,C 90.000,E1 276.947} C_DIS
LIN {X 0.009,Y -478.064,Z 331.534,A 0.000,B 0.000,C 90.000,E1 276.201} C_DIS
LIN {X 0.155,Y -480.515,Z 331.532,A 0.000,B 0.000,C 90.000,E1 275.682} C_DIS
LIN {X 0.135,Y -483.533,Z 331.527,A 0.000,B 0.000,C 90.000,E1 274.935} C_DIS
LIN {X -0.176,Y -485.069,Z 331.525,A 0.000,B 0.000,C 90.000,E1 274.473} C_DIS
LIN {X 0.004,Y -486.224,Z 331.522,A 0.000,B 0.000,C 90.000,E1 273.955} C_DIS
LIN {X 0.162,Y -486.911,Z 331.519,A 0.000,B 0.000,C 90.000,E1 273.440} C_DIS
LIN {X -0.131,Y -487.267,Z 331.516,A 0.000,B 0.000,C 90.000,E1 272.980} C_DIS
LIN {X 0.041,Y -487.332,Z 331.514,A 0.000,B 0.000,C 90.000,E1 272.465} C_DIS
LIN {X -0.076,Y -486.819,Z 331.508,A 0.000,B 0.000,C 90.000,E1 271.489} C_DIS
LIN {X 0.100,Y -486.355,Z 331.505,A 0.000,B 0.000,C 90.000,E1 270.974} C_DIS
LIN {X -0.210,Y -485.661,Z 331.503,A 0.000,B 0.000,C 90.000,E1 270.516} C_DIS
LIN {X -0.036,Y -484.627,Z 331.500,A 0.000,B 0.000,C 90.000,E1 270.000} C_DIS
LIN {X 0.133,Y -483.063,Z 331.497,A 0.000,B 0.000,C 90.000,E1 269.484} C_DIS
LIN {X -0.187,Y -480.914,Z 331.494,A 0.000,B 0.000,C 90.000,E1 269.026} C_DIS
LIN {X -0.035,Y -477.977,Z 331.492,A 0.000,B 0.000,C 90.000,E1 268.511} C_DIS
LIN {X -0.208,Y -476.203,Z 331.490,A 0.000,B 0.000,C 90.000,E1 268.282} C_DIS
LIN {X 0.109,Y -474.165,Z 331.489,A 0.000,B 0.000,C 90.000,E1 267.993} C_DIS
LIN {X 0.217,Y -469.211,Z 331.486,A 0.000,B 0.000,C 90.000,E1 267.478} C_DIS
LIN {X 0.120,Y -466.352,Z 331.485,A 0.000,B 0.000,C 90.000,E1 267.249} C_DIS
LIN {X 0.022,Y -463.131,Z 331.483,A 0.000,B 0.000,C 90.000,E1 267.020} C_DIS
LIN {X -0.217,Y -459.929,Z 331.482,A 0.000,B 0.000,C 90.000,E1 266.846} C_DIS
LIN {X 0.055,Y -452.877,Z 331.480,A 0.000,B 0.000,C 90.000,E1 266.445} C_DIS
LIN {X 0.038,Y -445.346,Z 331.479,A 0.000,B 0.000,C 90.000,E1 266.159} C_DIS
LIN {X 0.133,Y -437.431,Z 331.477,A 0.000,B 0.000,C 90.000,E1 265.927} C_DIS
LIN {X -0.175,Y -428.617,Z 331.477,A 0.000,B 0.000,C 90.000,E1 265.812} C_DIS
LIN {X -0.200,Y -421.865,Z 331.476,A 0.000,B 0.000,C 90.000,E1 265.755} C_DIS
LIN {X 0.095,Y -417.360,Z 331.476,A 0.000,B 0.000,C 90.000,E1 265.698} C_DIS
LIN {X 0.015,Y -180.911,Z 331.476,A 0.000,B 0.000,C 90.000,E1 265.698} C_DIS
LIN {X -0.061,Y -180.810,Z 331.471,A 0.000,B 0.000,C 90.000,E1 264.837} C_DIS
LIN {X 0.016,Y -178.913,Z 331.443,A 0.000,B 0.000,C 90.000,E1 259.746} C_DIS
LIN {X 0.095,Y -175.958,Z 331.415,A 0.000,B 0.000,C 90.000,E1 254.629} C_DIS
LIN {X 0.042,Y -175.428,Z 331.410,A 0.000,B 0.000,C 90.000,E1 253.795} C_DIS
LIN {X 0.045,Y -172.188,Z 331.386,A 0.000,B 0.000,C 90.000,E1 249.518} C_DIS
LIN {X 0.021,Y -171.660,Z 331.382,A 0.000,B 0.000,C 90.000,E1 248.666} C_DIS
LIN {X 0.005,Y -167.884,Z 331.358,A 0.000,B 0.000,C 90.000,E1 244.357} C_DIS
LIN {X 0.021,Y -166.622,Z 331.348,A 0.000,B 0.000,C 90.000,E1 242.615} C_DIS
LIN {X 0.014,Y -162.608,Z 331.324,A 0.000,B 0.000,C 90.000,E1 238.250} C_DIS
LIN {X -0.012,Y -161.294,Z 331.314,A 0.000,B 0.000,C 90.000,E1 236.501} C_DIS
LIN {X 0.022,Y -157.292,Z 331.289,A 0.000,B 0.000,C 90.000,E1 232.065} C_DIS
LIN {X 0.045,Y -156.008,Z 331.279,A 0.000,B 0.000,C 90.000,E1 230.275} C_DIS
LIN {X 0.005,Y -152.267,Z 331.255,A 0.000,B 0.000,C 90.000,E1 225.810} C_DIS
LIN {X 0.027,Y -150.504,Z 331.239,A 0.000,B 0.000,C 90.000,E1 223.095} C_DIS
LIN {X 0.056,Y -147.229,Z 331.214,A 0.000,B 0.000,C 90.000,E1 218.543} C_DIS
LIN {X 0.026,Y -145.251,Z 331.194,A 0.000,B 0.000,C 90.000,E1 214.898} C_DIS
LIN {X -0.058,Y -142.366,Z 331.163,A 0.000,B 0.000,C 90.000,E1 209.411} C_DIS
LIN {X 0.062,Y -141.752,Z 331.153,A 0.000,B 0.000,C 90.000,E1 207.513} C_DIS
LIN {X -0.011,Y -139.495,Z 331.117,A 0.000,B 0.000,C 90.000,E1 201.046} C_DIS
LIN {X 0.026,Y -139.000,Z 331.101,A 0.000,B 0.000,C 90.000,E1 198.236} C_DIS
LIN {X -0.018,Y -138.338,Z 331.055,A 0.000,B 0.000,C 90.000,E1 189.849} C_DIS
LIN {X 0.004,Y -139.411,Z 331.008,A 0.000,B 0.000,C 90.000,E1 181.432} C_DIS
LIN {X 0.057,Y -141.322,Z 330.972,A 0.000,B 0.000,C 90.000,E1 174.894} C_DIS
LIN {X 0.015,Y -142.680,Z 330.956,A 0.000,B 0.000,C 90.000,E1 172.129} C_DIS
LIN {X -0.005,Y -145.037,Z 330.931,A 0.000,B 0.000,C 90.000,E1 167.521} C_DIS
LIN {X -0.048,Y -147.662,Z 330.910,A 0.000,B 0.000,C 90.000,E1 163.866} C_DIS
LIN {X 0.028,Y -150.303,Z 330.890,A 0.000,B 0.000,C 90.000,E1 160.188} C_DIS
LIN {X 0.039,Y -153.712,Z 330.870,A 0.000,B 0.000,C 90.000,E1 156.561} C_DIS
LIN {X -0.048,Y -157.126,Z 330.850,A 0.000,B 0.000,C 90.000,E1 152.999} C_DIS
LIN {X 0.028,Y -161.271,Z 330.830,A 0.000,B 0.000,C 90.000,E1 149.410} C_DIS
LIN {X 0.046,Y -164.389,Z 330.815,A 0.000,B 0.000,C 90.000,E1 146.755} C_DIS
LIN {X 0.044,Y -169.066,Z 330.796,A 0.000,B 0.000,C 90.000,E1 143.256} C_DIS
LIN {X -0.006,Y -171.625,Z 330.786,A 0.000,B 0.000,C 90.000,E1 141.537} C_DIS
LIN {X 0.042,Y -176.584,Z 330.767,A 0.000,B 0.000,C 90.000,E1 138.081} C_DIS
LIN {X -0.085,Y -180.882,Z 330.753,A 0.000,B 0.000,C 90.000,E1 135.567} C_DIS
LIN {X 0.036,Y -186.297,Z 330.734,A 0.000,B 0.000,C 90.000,E1 132.162} C_DIS
LIN {X 0.103,Y -190.932,Z 330.720,A 0.000,B 0.000,C 90.000,E1 129.644} C_DIS
LIN {X 0.024,Y -196.700,Z 330.702,A 0.000,B 0.000,C 90.000,E1 126.377} C_DIS
LIN {X 0.000,Y -201.157,Z 330.690,A 0.000,B 0.000,C 90.000,E1 124.119} C_DIS
LIN {X -0.035,Y -301.896,Z 330.690,A 0.000,B 0.000,C 90.000,E1 124.119} C_DIS
LIN {X -0.140,Y -303.223,Z 330.689,A 0.000,B 0.000,C 90.000,E1 124.119} C_DIS
LIN {X 0.168,Y -306.999,Z 330.689,A 0.000,B 0.000,C 90.000,E1 123.913} C_DIS
LIN {X -0.049,Y -310.252,Z 330.687,A 0.000,B 0.000,C 90.000,E1 123.706} C_DIS
LIN {X 0.015,Y -313.954,Z 330.685,A 0.000,B 0.000,C 90.000,E1 123.245} C_DIS
LIN {X -0.194,Y -315.829,Z 330.683,A 0.000,B 0.000,C 90.000,E1 122.959} C_DIS
LIN {X -0.139,Y -317.299,Z 330.681,A 0.000,B 0.000,C 90.000,E1 122.625} C_DIS
LIN {X -0.002,Y -329.245,Z 330.663,A 0.000,B 0.000,C 90.000,E1 119.411} C_DIS
LIN {X -0.108,Y -341.404,Z 330.648,A 0.000,B 0.000,C 90.000,E1 116.616} C_DIS
LIN {X -0.044,Y -353.470,Z 330.634,A 0.000,B 0.000,C 90.000,E1 114.155} C_DIS
LIN {X 0.193,Y -366.809,Z 330.621,A 0.000,B 0.000,C 90.000,E1 111.716} C_DIS
LIN {X 0.016,Y -381.519,Z 330.608,A 0.000,B 0.000,C 90.000,E1 109.396} C_DIS
LIN {X 0.073,Y -397.708,Z 330.595,A 0.000,B 0.000,C 90.000,E1 107.094} C_DIS
LIN {X -0.100,Y -415.497,Z 330.583,A 0.000,B 0.000,C 90.000,E1 104.883} C_DIS
LIN {X 0.006,Y -434.936,Z 330.571,A 0.000,B 0.000,C 90.000,E1 102.703} C_DIS
LIN {X -0.169,Y -455.230,Z 330.559,A 0.000,B 0.000,C 90.000,E1 100.715} C_DIS
LIN {X -0.072,Y -476.055,Z 330.549,A 0.000,B 0.000,C 90.000,E1 98.859} C_DIS
LIN {X 0.080,Y -494.623,Z 330.541,A 0.000,B 0.000,C 90.000,E1 97.352} C_DIS
LIN {X -0.010,Y -498.348,Z 330.539,A 0.000,B 0.000,C 90.000,E1 96.947} C_DIS
LIN {X -0.161,Y -499.812,Z 330.537,A 0.000,B 0.000,C 90.000,E1 96.720} C_DIS
LIN {X 0.243,Y -500.900,Z 330.536,A 0.000,B 0.000,C 90.000,E1 96.429} C_DIS
LIN {X 0.028,Y -502.162,Z 330.533,A 0.000,B 0.000,C 90.000,E1 95.967} C_DIS
LIN {X -0.231,Y -502.385,Z 330.530,A 0.000,B 0.000,C 90.000,E1 95.511} C_DIS
LIN {X 0.068,Y -501.604,Z 330.528,A 0.000,B 0.000,C 90.000,E1 94.992} C_DIS
LIN {X -0.134,Y -499.681,Z 330.525,A 0.000,B 0.000,C 90.000,E1 94.531} C_DIS
LIN {X 0.154,Y -496.413,Z 330.522,A 0.000,B 0.000,C 90.000,E1 94.012} C_DIS
LIN {X -0.243,Y -490.854,Z 330.518,A 0.000,B 0.000,C 90.000,E1 93.326} C_DIS
LIN {X 0.173,Y -482.844,Z 330.513,A 0.000,B 0.000,C 90.000,E1 92.293} C_DIS
LIN {X -0.144,Y -458.842,Z 330.496,A 0.000,B 0.000,C 90.000,E1 89.312} C_DIS
LIN {X 0.017,Y -442.416,Z 330.483,A 0.000,B 0.000,C 90.000,E1 86.963} C_DIS
LIN {X 0.088,Y -424.174,Z 330.467,A 0.000,B 0.000,C 90.000,E1 84.033} C_DIS
LIN {X 0.150,Y -407.667,Z 330.450,A 0.000,B 0.000,C 90.000,E1 81.027} C_DIS
LIN {X 0.061,Y -396.182,Z 330.438,A 0.000,B 0.000,C 90.000,E1 78.814} C_DIS
LIN {X 0.068,Y -387.498,Z 330.428,A 0.000,B 0.000,C 90.000,E1 77.117} C_DIS
LIN {X 0.134,Y -375.833,Z 330.416,A 0.000,B 0.000,C 90.000,E1 74.810} C_DIS
LIN {X 0.043,Y -365.672,Z 330.404,A 0.000,B 0.000,C 90.000,E1 72.779} C_DIS
LIN {X -0.143,Y -355.476,Z 330.393,A 0.000,B 0.000,C 90.000,E1 70.732} C_DIS
LIN {X 0.059,Y -342.432,Z 330.378,A 0.000,B 0.000,C 90.000,E1 67.975} C_DIS
LIN {X -0.128,Y -331.648,Z 330.364,A 0.000,B 0.000,C 90.000,E1 65.537} C_DIS
LIN {X 0.121,Y -318.422,Z 330.345,A 0.000,B 0.000,C 90.000,E1 62.025} C_DIS
LIN {X 0.028,Y -307.095,Z 330.327,A 0.000,B 0.000,C 90.000,E1 58.820} C_DIS
LIN {X -0.022,Y -296.518,Z 330.309,A 0.000,B 0.000,C 90.000,E1 55.548} C_DIS
LIN {X 0.056,Y -286.652,Z 330.290,A 0.000,B 0.000,C 90.000,E1 52.190} C_DIS
LIN {X 0.114,Y -279.051,Z 330.275,A 0.000,B 0.000,C 90.000,E1 49.461} C_DIS
LIN {X 0.144,Y -273.296,Z 330.263,A 0.000,B 0.000,C 90.000,E1 47.391} C_DIS
LIN {X -0.002,Y -265.680,Z 330.248,A 0.000,B 0.000,C 90.000,E1 44.636} C_DIS
LIN {X -0.043,Y -260.043,Z 330.236,A 0.000,B 0.000,C 90.000,E1 42.528} C_DIS
LIN {X 0.007,Y -254.335,Z 330.224,A 0.000,B 0.000,C 90.000,E1 40.378} C_DIS
LIN {X -0.026,Y -248.601,Z 330.212,A 0.000,B 0.000,C 90.000,E1 38.222} C_DIS
LIN {X 0.071,Y -242.692,Z 330.200,A 0.000,B 0.000,C 90.000,E1 36.011} C_DIS
LIN {X -0.070,Y -234.861,Z 330.184,A 0.000,B 0.000,C 90.000,E1 33.086} C_DIS
LIN {X -0.062,Y -227.316,Z 330.167,A 0.000,B 0.000,C 90.000,E1 30.079} C_DIS
LIN {X 0.040,Y -220.194,Z 330.150,A 0.000,B 0.000,C 90.000,E1 27.001} C_DIS
LIN {X 0.056,Y -213.726,Z 330.133,A 0.000,B 0.000,C 90.000,E1 23.898} C_DIS
LIN {X -0.063,Y -208.120,Z 330.115,A 0.000,B 0.000,C 90.000,E1 20.791} C_DIS
LIN {X -0.027,Y -202.126,Z 330.093,A 0.000,B 0.000,C 90.000,E1 16.804} C_DIS
LIN {X -0.049,Y -198.082,Z 330.075,A 0.000,B 0.000,C 90.000,E1 13.592} C_DIS
LIN {X 0.051,Y -194.139,Z 330.053,A 0.000,B 0.000,C 90.000,E1 9.500} C_DIS
LIN {X 0.031,Y -190.826,Z 330.026,A 0.000,B 0.000,C 90.000,E1 4.588} C_DIS
LIN {X -0.096,Y -188.682,Z 329.984,A 0.000,B 0.000,C 90.000,E1 357.078} C_DIS
LIN {X 0.027,Y -190.593,Z 329.933,A 0.000,B 0.000,C 90.000,E1 347.937} C_DIS
LIN {X -0.031,Y -193.780,Z 329.906,A 0.000,B 0.000,C 90.000,E1 343.015} C_DIS
LIN {X 0.063,Y -197.633,Z 329.883,A 0.000,B 0.000,C 90.000,E1 338.901} C_DIS
LIN {X 0.085,Y -202.496,Z 329.860,A 0.000,B 0.000,C 90.000,E1 334.845} C_DIS
LIN {X 0.065,Y -208.356,Z 329.838,A 0.000,B 0.000,C 90.000,E1 330.845} C_DIS
LIN {X -0.014,Y -215.214,Z 329.816,A 0.000,B 0.000,C 90.000,E1 326.914} C_DIS
LIN {X 0.045,Y -222.780,Z 329.795,A 0.000,B 0.000,C 90.000,E1 323.004} C_DIS
LIN {X 0.148,Y -229.511,Z 329.777,A 0.000,B 0.000,C 90.000,E1 319.908} C_DIS
LIN {X 0.021,Y -238.203,Z 329.759,A 0.000,B 0.000,C 90.000,E1 316.539} C_DIS
LIN {X -0.030,Y -248.384,Z 329.740,A 0.000,B 0.000,C 90.000,E1 313.218} C_DIS
LIN {X 0.079,Y -259.641,Z 329.722,A 0.000,B 0.000,C 90.000,E1 309.930} C_DIS
LIN {X 0.057,Y -271.800,Z 329.704,A 0.000,B 0.000,C 90.000,E1 306.744} C_DIS
LIN {X -0.106,Y -280.653,Z 329.693,A 0.000,B 0.000,C 90.000,E1 304.692} C_DIS
LIN {X 0.086,Y -293.582,Z 329.677,A 0.000,B 0.000,C 90.000,E1 301.926} C_DIS
LIN {X 0.032,Y -309.641,Z 329.661,A 0.000,B 0.000,C 90.000,E1 298.949} C_DIS
LIN {X -0.018,Y -319.335,Z 329.652,A 0.000,B 0.000,C 90.000,E1 297.334} C_DIS
LIN {X 0.102,Y -338.537,Z 329.636,A 0.000,B 0.000,C 90.000,E1 294.463} C_DIS
END
